LIN {X 0,Y 688.4,Z 749.56,A -85,B 0,C 180,E1 4160.047,E2 4160.047} C_VEL
LIN {X 0,Y 687.145,Z 749.56,A -85,B 0,C 180,E1 4160.767,E2 4160.767} C_VEL
LIN {X 0,Y 680.483,Z 749.56,A -85,B 0,C 180,E1 4162.72,E2 4162.72} C_VEL
LIN {X 0,Y 680.39,Z 749.56,A -85,B 0,C 180,E1 4162.905,E2 4162.905} C_VEL
LIN {X 0,Y 680.421,Z 749.56,A -85,B 0,C 180,E1 4167.797,E2 4167.797} C_VEL
LIN {X 0,Y 680.331,Z 749.56,A -85,B 0,C 180,E1 4172.429,E2 4172.429} C_VEL
LIN {X 0,Y 680.255,Z 749.56,A -85,B 0,C 180,E1 4176.897,E2 4176.897} C_VEL
LIN {X 0,Y 680.389,Z 749.56,A -85,B 0,C 180,E1 4182.867,E2 4182.867} C_VEL
LIN {X 0,Y 680.257,Z 749.803,A -85,B 0,C 180,E1 4188.162,E2 4188.162} C_VEL
LIN {X 0,Y 684.994,Z 759.606,A -85,B 0,C 180,E1 4188.65,E2 4188.65} C_VEL
LIN {X 0,Y 698.353,Z 783.089,A -85,B 0,C 180,E1 4189.918,E2 4189.918} C_VEL
LIN {X 0,Y 697.598,Z 850.093,A -85,B 0,C 180,E1 4190.892,E2 4190.892} C_VEL
LIN {X 0,Y 695.833,Z 894.125,A -85,B 0,C 180,E1 4191.958,E2 4191.958} C_VEL
LIN {X 0,Y 693.647,Z 941.776,A -85,B 0,C 180,E1 4193.674,E2 4193.674} C_VEL
LIN {X 0,Y 691.134,Z 988.011,A -85,B 0,C 180,E1 4195.911,E2 4195.911} C_VEL
LIN {X 0,Y 688.572,Z 1030.029,A -85,B 0,C 180,E1 4198.54,E2 4198.54} C_VEL
LIN {X 0,Y 686.252,Z 1069.067,A -85,B 0,C 180,E1 4201.577,E2 4201.577} C_VEL
LIN {X 0,Y 684.111,Z 1106.115,A -85,B 0,C 180,E1 4205.184,E2 4205.184} C_VEL
LIN {X 0,Y 682.717,Z 1135.913,A -85,B 0,C 180,E1 4208.795,E2 4208.795} C_VEL
LIN {X 0,Y 681.777,Z 1162.143,A -85,B 0,C 180,E1 4212.802,E2 4212.802} C_VEL
LIN {X 0,Y 681.145,Z 1182.346,A -85,B 0,C 180,E1 4216.855,E2 4216.855} C_VEL
LIN {X 0,Y 680.941,Z 1196.276,A -85,B 0,C 180,E1 4220.7,E2 4220.7} C_VEL
LIN {X 0,Y 680.837,Z 1204.797,A -85,B 0,C 180,E1 4224.267,E2 4224.267} C_VEL
LIN {X 0,Y 680.8,Z 1208.952,A -85,B 0,C 180,E1 4227.455,E2 4227.455} C_VEL
LIN {X 0,Y 680.945,Z 1209.669,A -85,B 0,C 180,E1 4231.271,E2 4231.271} C_VEL
LIN {X 0,Y 680.757,Z 1205.912,A -85,B 0,C 180,E1 4235.093,E2 4235.093} C_VEL
LIN {X 0,Y 680.821,Z 1197.333,A -85,B 0,C 180,E1 4238.938,E2 4238.938} C_VEL
LIN {X 0,Y 680.999,Z 1185.052,A -85,B 0,C 180,E1 4242.495,E2 4242.495} C_VEL
LIN {X 0,Y 681.502,Z 1166.472,A -85,B 0,C 180,E1 4246.421,E2 4246.421} C_VEL
LIN {X 0,Y 682.336,Z 1143.81,A -85,B 0,C 180,E1 4250.111,E2 4250.111} C_VEL
LIN {X 0,Y 683.774,Z 1113.746,A -85,B 0,C 180,E1 4253.958,E2 4253.958} C_VEL
LIN {X 0,Y 685.541,Z 1080.468,A -85,B 0,C 180,E1 4257.394,E2 4257.394} C_VEL
LIN {X 0,Y 687.949,Z 1040.284,A -85,B 0,C 180,E1 4260.73,E2 4260.73} C_VEL
LIN {X 0,Y 690.402,Z 998.657,A -85,B 0,C 180,E1 4263.478,E2 4263.478} C_VEL
LIN {X 0,Y 693.13,Z 953.433,A -85,B 0,C 180,E1 4265.821,E2 4265.821} C_VEL
LIN {X 0,Y 695.261,Z 909.712,A -85,B 0,C 180,E1 4267.534,E2 4267.534} C_VEL
LIN {X 0,Y 696.967,Z 867.67,A -85,B 0,C 180,E1 4268.733,E2 4268.733} C_VEL
LIN {X 0,Y 698.111,Z 822.718,A -85,B 0,C 180,E1 4269.568,E2 4269.568} C_VEL
LIN {X 0,Y 697.756,Z 782.473,A -85,B 0,C 180,E1 4270.132,E2 4270.132} C_VEL
LIN {X 0,Y 680.589,Z 751.281,A -85,B 0,C 180,E1 4271.792,E2 4271.792} C_VEL
LIN {X 0,Y 680.389,Z 749.56,A -85,B 0,C 180,E1 4271.887,E2 4271.887} C_VEL
LIN {X 0,Y 680.266,Z 749.56,A -85,B 0,C 180,E1 4276.482,E2 4276.482} C_VEL
LIN {X 0,Y 680.222,Z 749.56,A -85,B 0,C 180,E1 4281.539,E2 4281.539} C_VEL
LIN {X 0,Y 680.183,Z 749.56,A -85,B 0,C 180,E1 4286.264,E2 4286.264} C_VEL
LIN {X 0,Y 680.22,Z 749.56,A -85,B 0,C 180,E1 4290.746,E2 4290.746} C_VEL
LIN {X 0,Y 680.282,Z 749.56,A -85,B 0,C 180,E1 4295.607,E2 4295.607} C_VEL
LIN {X 0,Y 680.357,Z 749.56,A -85,B 0,C 180,E1 4300.542,E2 4300.542} C_VEL
LIN {X 0,Y 680.522,Z 749.56,A -85,B 0,C 180,E1 4305.865,E2 4305.865} C_VEL
LIN {X 0,Y 680.663,Z 749.56,A -85,B 0,C 180,E1 4311.063,E2 4311.063} C_VEL
LIN {X 0,Y 680.71,Z 749.56,A -85,B 0,C 180,E1 4316.185,E2 4316.185} C_VEL
LIN {X 0,Y 680.718,Z 749.56,A -85,B 0,C 180,E1 4320.004,E2 4320.004} C_VEL
LIN {X 0,Y 680.625,Z 749.56,A -85,B 0,C 180,E1 4325.099,E2 4325.099} C_VEL
LIN {X 0,Y 680.622,Z 749.56,A -85,B 0,C 180,E1 4330.235,E2 4330.235} C_VEL
LIN {X 0,Y 680.3,Z 749.56,A -85,B 0,C 180,E1 4335.463,E2 4335.463} C_VEL
LIN {X 0,Y 680.262,Z 749.56,A -85,B 0,C 180,E1 4341.097,E2 4341.097} C_VEL
LIN {X 0,Y 680.207,Z 749.56,A -85,B 0,C 180,E1 4346.384,E2 4346.384} C_VEL
LIN {X 0,Y 680.221,Z 749.56,A -85,B 0,C 180,E1 4350.732,E2 4350.732} C_VEL
LIN {X 0,Y 680.223,Z 749.56,A -85,B 0,C 180,E1 4355.287,E2 4355.287} C_VEL
LIN {X 0,Y 680.229,Z 749.56,A -85,B 0,C 180,E1 4360.114,E2 4360.114} C_VEL
LIN {X 0,Y 680.28,Z 749.714,A -85,B 0,C 180,E1 4363.859,E2 4363.859} C_VEL
LIN {X 0,Y 687.051,Z 763.886,A -85,B 0,C 180,E1 4364.465,E2 4364.465} C_VEL
LIN {X 0,Y 694.991,Z 780.667,A -85,B 0,C 180,E1 4365.184,E2 4365.184} C_VEL
LIN {X 0,Y 693.799,Z 827.247,A -85,B 0,C 180,E1 4366.107,E2 4366.107} C_VEL
LIN {X 0,Y 692.079,Z 873.368,A -85,B 0,C 180,E1 4367.568,E2 4367.568} C_VEL
LIN {X 0,Y 689.888,Z 916.339,A -85,B 0,C 180,E1 4369.457,E2 4369.457} C_VEL
LIN {X 0,Y 687.699,Z 958.747,A -85,B 0,C 180,E1 4371.915,E2 4371.915} C_VEL
LIN {X 0,Y 685.492,Z 998.587,A -85,B 0,C 180,E1 4374.891,E2 4374.891} C_VEL
LIN {X 0,Y 683.747,Z 1032.734,A -85,B 0,C 180,E1 4378.117,E2 4378.117} C_VEL
LIN {X 0,Y 682.43,Z 1061.896,A -85,B 0,C 180,E1 4381.571,E2 4381.571} C_VEL
LIN {X 0,Y 681.515,Z 1087.051,A -85,B 0,C 180,E1 4385.392,E2 4385.392} C_VEL
LIN {X 0,Y 681.141,Z 1103.808,A -85,B 0,C 180,E1 4388.727,E2 4388.727} C_VEL
LIN {X 0,Y 680.802,Z 1117.989,A -85,B 0,C 180,E1 4392.655,E2 4392.655} C_VEL
LIN {X 0,Y 680.792,Z 1125.467,A -85,B 0,C 180,E1 4395.868,E2 4395.868} C_VEL
LIN {X 0,Y 680.667,Z 1129.693,A -85,B 0,C 180,E1 4399.77,E2 4399.77} C_VEL
LIN {X 0,Y 680.816,Z 1128.697,A -85,B 0,C 180,E1 4403.629,E2 4403.629} C_VEL
LIN {X 0,Y 680.837,Z 1122.652,A -85,B 0,C 180,E1 4407.456,E2 4407.456} C_VEL
LIN {X 0,Y 680.918,Z 1111.397,A -85,B 0,C 180,E1 4411.272,E2 4411.272} C_VEL
LIN {X 0,Y 681.281,Z 1096.404,A -85,B 0,C 180,E1 4414.772,E2 4414.772} C_VEL
LIN {X 0,Y 681.915,Z 1075.181,A -85,B 0,C 180,E1 4418.443,E2 4418.443} C_VEL
LIN {X 0,Y 682.954,Z 1049.025,A -85,B 0,C 180,E1 4421.973,E2 4421.973} C_VEL
LIN {X 0,Y 684.646,Z 1014.871,A -85,B 0,C 180,E1 4425.577,E2 4425.577} C_VEL
LIN {X 0,Y 686.685,Z 976.797,A -85,B 0,C 180,E1 4428.732,E2 4428.732} C_VEL
LIN {X 0,Y 688.86,Z 937.867,A -85,B 0,C 180,E1 4431.278,E2 4431.278} C_VEL
LIN {X 0,Y 691.074,Z 895.773,A -85,B 0,C 180,E1 4433.426,E2 4433.426} C_VEL
LIN {X 0,Y 692.994,Z 852.505,A -85,B 0,C 180,E1 4435.065,E2 4435.065} C_VEL
LIN {X 0,Y 694.484,Z 807.428,A -85,B 0,C 180,E1 4436.259,E2 4436.259} C_VEL
LIN {X 0,Y 694.58,Z 779.374,A -85,B 0,C 180,E1 4436.77,E2 4436.77} C_VEL
LIN {X 0,Y 680.489,Z 750.957,A -85,B 0,C 180,E1 4438.022,E2 4438.022} C_VEL
LIN {X 0,Y 680.342,Z 749.56,A -85,B 0,C 180,E1 4438.085,E2 4438.085} C_VEL
LIN {X 0,Y 680.265,Z 749.56,A -85,B 0,C 180,E1 4443.735,E2 4443.735} C_VEL
LIN {X 0,Y 680.155,Z 749.56,A -85,B 0,C 180,E1 4448.951,E2 4448.951} C_VEL
LIN {X 0,Y 680.399,Z 749.56,A -85,B 0,C 180,E1 4453.512,E2 4453.512} C_VEL
LIN {X 0,Y 680.181,Z 749.56,A -85,B 0,C 180,E1 4459.058,E2 4459.058} C_VEL
LIN {X 0,Y 680.219,Z 749.56,A -85,B 0,C 180,E1 4463.138,E2 4463.138} C_VEL
LIN {X 0,Y 680.157,Z 749.56,A -85,B 0,C 180,E1 4467.772,E2 4467.772} C_VEL
LIN {X 0,Y 680.239,Z 749.56,A -85,B 0,C 180,E1 4472.698,E2 4472.698} C_VEL
LIN {X 0,Y 680.175,Z 749.56,A -85,B 0,C 180,E1 4477.805,E2 4477.805} C_VEL
LIN {X 0,Y 680.129,Z 749.56,A -85,B 0,C 180,E1 4482.823,E2 4482.823} C_VEL
LIN {X 0,Y 680.461,Z 749.56,A -85,B 0,C 180,E1 4487.724,E2 4487.724} C_VEL
LIN {X 0,Y 680.693,Z 749.56,A -85,B 0,C 180,E1 4492.342,E2 4492.342} C_VEL
LIN {X 0,Y 680.789,Z 749.56,A -85,B 0,C 180,E1 4497.452,E2 4497.452} C_VEL
LIN {X 0,Y 680.649,Z 749.56,A -85,B 0,C 180,E1 4502.541,E2 4502.541} C_VEL
LIN {X 0,Y 680.615,Z 749.56,A -85,B 0,C 180,E1 4506.37,E2 4506.37} C_VEL
LIN {X 0,Y 680.53,Z 749.56,A -85,B 0,C 180,E1 4511.525,E2 4511.525} C_VEL
LIN {X 0,Y 680.581,Z 749.56,A -85,B 0,C 180,E1 4516.774,E2 4516.774} C_VEL
LIN {X 0,Y 680.445,Z 749.56,A -85,B 0,C 180,E1 4522.178,E2 4522.178} C_VEL
LIN {X 0,Y 680.39,Z 749.56,A -85,B 0,C 180,E1 4522.905,E2 4522.905} C_VEL
LIN {X 0,Y 676.44,Z 749.56,A -85,B 0,C 180,E1 4524.339,E2 4524.339} C_VEL
LIN {X 0,Y 672.491,Z 749.56,A -85,B 0,C 180,E1 4525.789,E2 4525.789} C_VEL
LIN {X 0,Y 672.379,Z 749.56,A -85,B 0,C 180,E1 4531.347,E2 4531.347} C_VEL
LIN {X 0,Y 672.337,Z 749.56,A -85,B 0,C 180,E1 4535.988,E2 4535.988} C_VEL
LIN {X 0,Y 672.281,Z 749.56,A -85,B 0,C 180,E1 4540.678,E2 4540.678} C_VEL
LIN {X 0,Y 672.404,Z 749.56,A -85,B 0,C 180,E1 4545.981,E2 4545.981} C_VEL
LIN {X 0,Y 672.318,Z 749.803,A -85,B 0,C 180,E1 4547.554,E2 4547.554} C_VEL
LIN {X 0,Y 674.866,Z 755.349,A -85,B 0,C 180,E1 4547.829,E2 4547.829} C_VEL
LIN {X 0,Y 692.164,Z 785.898,A -85,B 0,C 180,E1 4549.523,E2 4549.523} C_VEL
LIN {X 0,Y 691.411,Z 851.6,A -85,B 0,C 180,E1 4550.506,E2 4550.506} C_VEL
LIN {X 0,Y 689.52,Z 895.054,A -85,B 0,C 180,E1 4551.576,E2 4551.576} C_VEL
LIN {X 0,Y 687.082,Z 942.72,A -85,B 0,C 180,E1 4553.314,E2 4553.314} C_VEL
LIN {X 0,Y 684.338,Z 988.281,A -85,B 0,C 180,E1 4555.54,E2 4555.54} C_VEL
LIN {X 0,Y 681.494,Z 1030.32,A -85,B 0,C 180,E1 4558.197,E2 4558.197} C_VEL
LIN {X 0,Y 678.955,Z 1069.071,A -85,B 0,C 180,E1 4561.243,E2 4561.243} C_VEL
LIN {X 0,Y 676.611,Z 1106.113,A -85,B 0,C 180,E1 4564.89,E2 4564.89} C_VEL
LIN {X 0,Y 675.023,Z 1136.317,A -85,B 0,C 180,E1 4568.598,E2 4568.598} C_VEL
LIN {X 0,Y 673.984,Z 1162.44,A -85,B 0,C 180,E1 4572.648,E2 4572.648} C_VEL
LIN {X 0,Y 673.306,Z 1182.347,A -85,B 0,C 180,E1 4576.7,E2 4576.7} C_VEL
LIN {X 0,Y 673.083,Z 1195.433,A -85,B 0,C 180,E1 4580.306,E2 4580.306} C_VEL
LIN {X 0,Y 672.955,Z 1204.795,A -85,B 0,C 180,E1 4584.2,E2 4584.2} C_VEL
LIN {X 0,Y 672.921,Z 1208.949,A -85,B 0,C 180,E1 4587.425,E2 4587.425} C_VEL
LIN {X 0,Y 673.045,Z 1209.669,A -85,B 0,C 180,E1 4591.286,E2 4591.286} C_VEL
LIN {X 0,Y 672.859,Z 1205.912,A -85,B 0,C 180,E1 4595.153,E2 4595.153} C_VEL
LIN {X 0,Y 672.96,Z 1197.333,A -85,B 0,C 180,E1 4599.043,E2 4599.043} C_VEL
LIN {X 0,Y 673.171,Z 1183.704,A -85,B 0,C 180,E1 4602.972,E2 4602.972} C_VEL
LIN {X 0,Y 673.827,Z 1164.715,A -85,B 0,C 180,E1 4606.949,E2 4606.949} C_VEL
LIN {X 0,Y 674.869,Z 1139.247,A -85,B 0,C 180,E1 4610.993,E2 4610.993} C_VEL
LIN {X 0,Y 676.475,Z 1109.315,A -85,B 0,C 180,E1 4614.761,E2 4614.761} C_VEL
LIN {X 0,Y 678.707,Z 1072.626,A -85,B 0,C 180,E1 4618.432,E2 4618.432} C_VEL
LIN {X 0,Y 681.195,Z 1035.134,A -85,B 0,C 180,E1 4621.46,E2 4621.46} C_VEL
LIN {X 0,Y 684.014,Z 991.951,A -85,B 0,C 180,E1 4624.252,E2 4624.252} C_VEL
LIN {X 0,Y 686.772,Z 948.289,A -85,B 0,C 180,E1 4626.447,E2 4626.447} C_VEL
LIN {X 0,Y 689.265,Z 900.278,A -85,B 0,C 180,E1 4628.256,E2 4628.256} C_VEL
LIN {X 0,Y 691.183,Z 852.976,A -85,B 0,C 180,E1 4629.48,E2 4629.48} C_VEL
LIN {X 0,Y 691.817,Z 785.747,A -85,B 0,C 180,E1 4630.504,E2 4630.504} C_VEL
LIN {X 0,Y 672.601,Z 751.041,A -85,B 0,C 180,E1 4632.407,E2 4632.407} C_VEL
LIN {X 0,Y 672.492,Z 749.56,A -85,B 0,C 180,E1 4632.493,E2 4632.493} C_VEL
LIN {X 0,Y 672.272,Z 749.56,A -85,B 0,C 180,E1 4637.882,E2 4637.882} C_VEL
LIN {X 0,Y 672.298,Z 749.56,A -85,B 0,C 180,E1 4642.639,E2 4642.639} C_VEL
LIN {X 0,Y 672.266,Z 749.56,A -85,B 0,C 180,E1 4647.355,E2 4647.355} C_VEL
LIN {X 0,Y 672.32,Z 749.56,A -85,B 0,C 180,E1 4651.839,E2 4651.839} C_VEL
LIN {X 0,Y 672.333,Z 749.56,A -85,B 0,C 180,E1 4657.146,E2 4657.146} C_VEL
LIN {X 0,Y 672.476,Z 749.56,A -85,B 0,C 180,E1 4661.667,E2 4661.667} C_VEL
LIN {X 0,Y 672.663,Z 749.56,A -85,B 0,C 180,E1 4667.021,E2 4667.021} C_VEL
LIN {X 0,Y 672.723,Z 749.56,A -85,B 0,C 180,E1 4672.258,E2 4672.258} C_VEL
LIN {X 0,Y 672.808,Z 749.56,A -85,B 0,C 180,E1 4676.14,E2 4676.14} C_VEL
LIN {X 0,Y 672.823,Z 749.56,A -85,B 0,C 180,E1 4680.004,E2 4680.004} C_VEL
LIN {X 0,Y 672.827,Z 749.56,A -85,B 0,C 180,E1 4683.867,E2 4683.867} C_VEL
LIN {X 0,Y 672.684,Z 749.56,A -85,B 0,C 180,E1 4689.051,E2 4689.051} C_VEL
LIN {X 0,Y 672.465,Z 749.56,A -85,B 0,C 180,E1 4694.315,E2 4694.315} C_VEL
LIN {X 0,Y 672.38,Z 749.56,A -85,B 0,C 180,E1 4699.705,E2 4699.705} C_VEL
LIN {X 0,Y 672.257,Z 749.56,A -85,B 0,C 180,E1 4705.288,E2 4705.288} C_VEL
LIN {X 0,Y 672.301,Z 749.56,A -85,B 0,C 180,E1 4709.641,E2 4709.641} C_VEL
LIN {X 0,Y 672.296,Z 749.56,A -85,B 0,C 180,E1 4714.194,E2 4714.194} C_VEL
LIN {X 0,Y 672.345,Z 749.56,A -85,B 0,C 180,E1 4719.005,E2 4719.005} C_VEL
LIN {X 0,Y 672.312,Z 749.56,A -85,B 0,C 180,E1 4723.34,E2 4723.34} C_VEL
LIN {X 0,Y 676.815,Z 759.567,A -85,B 0,C 180,E1 4723.765,E2 4723.765} C_VEL
LIN {X 0,Y 688.564,Z 782.52,A -85,B 0,C 180,E1 4724.825,E2 4724.825} C_VEL
LIN {X 0,Y 687.23,Z 828.392,A -85,B 0,C 180,E1 4725.759,E2 4725.759} C_VEL
LIN {X 0,Y 685.332,Z 874.495,A -85,B 0,C 180,E1 4727.239,E2 4727.239} C_VEL
LIN {X 0,Y 682.895,Z 917.839,A -85,B 0,C 180,E1 4729.179,E2 4729.179} C_VEL
LIN {X 0,Y 680.516,Z 959.618,A -85,B 0,C 180,E1 4731.642,E2 4731.642} C_VEL
LIN {X 0,Y 678.036,Z 1000.415,A -85,B 0,C 180,E1 4734.738,E2 4734.738} C_VEL
LIN {X 0,Y 676.02,Z 1035.648,A -85,B 0,C 180,E1 4738.158,E2 4738.158} C_VEL
LIN {X 0,Y 674.614,Z 1064.21,A -85,B 0,C 180,E1 4741.661,E2 4741.661} C_VEL
LIN {X 0,Y 673.684,Z 1088.271,A -85,B 0,C 180,E1 4745.42,E2 4745.42} C_VEL
LIN {X 0,Y 673.17,Z 1106.738,A -85,B 0,C 180,E1 4749.296,E2 4749.296} C_VEL
LIN {X 0,Y 672.881,Z 1119.377,A -85,B 0,C 180,E1 4753.026,E2 4753.026} C_VEL
LIN {X 0,Y 672.845,Z 1126.427,A -85,B 0,C 180,E1 4756.361,E2 4756.361} C_VEL
LIN {X 0,Y 672.771,Z 1129.664,A -85,B 0,C 180,E1 4759.649,E2 4759.649} C_VEL
LIN {X 0,Y 672.909,Z 1128.781,A -85,B 0,C 180,E1 4763.554,E2 4763.554} C_VEL
LIN {X 0,Y 672.968,Z 1122.908,A -85,B 0,C 180,E1 4767.427,E2 4767.427} C_VEL
LIN {X 0,Y 673.046,Z 1111.775,A -85,B 0,C 180,E1 4771.287,E2 4771.287} C_VEL
LIN {X 0,Y 673.417,Z 1096.913,A -85,B 0,C 180,E1 4774.828,E2 4774.828} C_VEL
LIN {X 0,Y 674.114,Z 1075.897,A -85,B 0,C 180,E1 4778.541,E2 4778.541} C_VEL
LIN {X 0,Y 675.248,Z 1049.936,A -85,B 0,C 180,E1 4782.111,E2 4782.111} C_VEL
LIN {X 0,Y 677.043,Z 1017.091,A -85,B 0,C 180,E1 4785.65,E2 4785.65} C_VEL
LIN {X 0,Y 679.171,Z 981.604,A -85,B 0,C 180,E1 4788.689,E2 4788.689} C_VEL
LIN {X 0,Y 681.648,Z 942.01,A -85,B 0,C 180,E1 4791.382,E2 4791.382} C_VEL
LIN {X 0,Y 684.033,Z 899.754,A -85,B 0,C 180,E1 4793.604,E2 4793.604} C_VEL
LIN {X 0,Y 686.094,Z 858.301,A -85,B 0,C 180,E1 4795.257,E2 4795.257} C_VEL
LIN {X 0,Y 687.88,Z 810.271,A -85,B 0,C 180,E1 4796.579,E2 4796.579} C_VEL
LIN {X 0,Y 688.21,Z 782.176,A -85,B 0,C 180,E1 4797.111,E2 4797.111} C_VEL
LIN {X 0,Y 672.466,Z 749.56,A -85,B 0,C 180,E1 4798.591,E2 4798.591} C_VEL
LIN {X 0,Y 672.361,Z 749.56,A -85,B 0,C 180,E1 4804.186,E2 4804.186} C_VEL
LIN {X 0,Y 672.263,Z 749.56,A -85,B 0,C 180,E1 4809.006,E2 4809.006} C_VEL
LIN {X 0,Y 672.472,Z 749.56,A -85,B 0,C 180,E1 4814.156,E2 4814.156} C_VEL
LIN {X 0,Y 672.343,Z 749.56,A -85,B 0,C 180,E1 4819.834,E2 4819.834} C_VEL
LIN {X 0,Y 672.271,Z 749.56,A -85,B 0,C 180,E1 4824.232,E2 4824.232} C_VEL
LIN {X 0,Y 672.243,Z 749.56,A -85,B 0,C 180,E1 4828.863,E2 4828.863} C_VEL
LIN {X 0,Y 672.275,Z 749.56,A -85,B 0,C 180,E1 4834.043,E2 4834.043} C_VEL
LIN {X 0,Y 672.343,Z 749.56,A -85,B 0,C 180,E1 4838.919,E2 4838.919} C_VEL
LIN {X 0,Y 672.385,Z 749.56,A -85,B 0,C 180,E1 4844.35,E2 4844.35} C_VEL
LIN {X 0,Y 672.729,Z 749.56,A -85,B 0,C 180,E1 4849.644,E2 4849.644} C_VEL
LIN {X 0,Y 672.728,Z 749.56,A -85,B 0,C 180,E1 4854.841,E2 4854.841} C_VEL
LIN {X 0,Y 672.851,Z 749.56,A -85,B 0,C 180,E1 4859.996,E2 4859.996} C_VEL
LIN {X 0,Y 672.882,Z 749.56,A -85,B 0,C 180,E1 4865.15,E2 4865.15} C_VEL
LIN {X 0,Y 672.67,Z 749.56,A -85,B 0,C 180,E1 4870.35,E2 4870.35} C_VEL
LIN {X 0,Y 672.661,Z 749.56,A -85,B 0,C 180,E1 4875.636,E2 4875.636} C_VEL
LIN {X 0,Y 672.594,Z 749.56,A -85,B 0,C 180,E1 4881.065,E2 4881.065} C_VEL
LIN {X 0,Y 672.491,Z 749.56,A -85,B 0,C 180,E1 4885.789,E2 4885.789} C_VEL
LIN {X 0,Y 671.256,Z 749.56,A -85,B 0,C 180,E1 4886.527,E2 4886.527} C_VEL
LIN {X 0,Y 664.616,Z 749.56,A -85,B 0,C 180,E1 4888.532,E2 4888.532} C_VEL
LIN {X 0,Y 664.498,Z 749.56,A -85,B 0,C 180,E1 4888.721,E2 4888.721} C_VEL
LIN {X 0,Y 664.529,Z 749.56,A -85,B 0,C 180,E1 4893.073,E2 4893.073} C_VEL
LIN {X 0,Y 664.37,Z 749.56,A -85,B 0,C 180,E1 4897.885,E2 4897.885} C_VEL
LIN {X 0,Y 664.493,Z 749.56,A -85,B 0,C 180,E1 4903.304,E2 4903.304} C_VEL
LIN {X 0,Y 664.428,Z 749.803,A -85,B 0,C 180,E1 4906.928,E2 4906.928} C_VEL
LIN {X 0,Y 667.032,Z 755.395,A -85,B 0,C 180,E1 4907.217,E2 4907.217} C_VEL
LIN {X 0,Y 686.149,Z 789.017,A -85,B 0,C 180,E1 4909.135,E2 4909.135} C_VEL
LIN {X 0,Y 685.237,Z 852.824,A -85,B 0,C 180,E1 4910.106,E2 4910.106} C_VEL
LIN {X 0,Y 683.131,Z 897.169,A -85,B 0,C 180,E1 4911.225,E2 4911.225} C_VEL
LIN {X 0,Y 680.403,Z 945.663,A -85,B 0,C 180,E1 4913.032,E2 4913.032} C_VEL
LIN {X 0,Y 677.474,Z 989.991,A -85,B 0,C 180,E1 4915.247,E2 4915.247} C_VEL
LIN {X 0,Y 674.297,Z 1033.297,A -85,B 0,C 180,E1 4918.042,E2 4918.042} C_VEL
LIN {X 0,Y 671.543,Z 1071.067,A -85,B 0,C 180,E1 4921.087,E2 4921.087} C_VEL
LIN {X 0,Y 668.981,Z 1108.342,A -85,B 0,C 180,E1 4924.834,E2 4924.834} C_VEL
LIN {X 0,Y 667.246,Z 1138.185,A -85,B 0,C 180,E1 4928.603,E2 4928.603} C_VEL
LIN {X 0,Y 666.176,Z 1163.173,A -85,B 0,C 180,E1 4932.567,E2 4932.567} C_VEL
LIN {X 0,Y 665.489,Z 1182.348,A -85,B 0,C 180,E1 4936.54,E2 4936.54} C_VEL
LIN {X 0,Y 665.216,Z 1195.43,A -85,B 0,C 180,E1 4940.19,E2 4940.19} C_VEL
LIN {X 0,Y 665.075,Z 1204.793,A -85,B 0,C 180,E1 4944.131,E2 4944.131} C_VEL
LIN {X 0,Y 665.017,Z 1208.946,A -85,B 0,C 180,E1 4947.395,E2 4947.395} C_VEL
LIN {X 0,Y 665.128,Z 1209.591,A -85,B 0,C 180,E1 4951.594,E2 4951.594} C_VEL
LIN {X 0,Y 665.034,Z 1204.796,A -85,B 0,C 180,E1 4955.868,E2 4955.868} C_VEL
LIN {X 0,Y 665.252,Z 1194.434,A -85,B 0,C 180,E1 4960.139,E2 4960.139} C_VEL
LIN {X 0,Y 665.566,Z 1179.548,A -85,B 0,C 180,E1 4964.126,E2 4964.126} C_VEL
LIN {X 0,Y 666.342,Z 1158.242,A -85,B 0,C 180,E1 4968.288,E2 4968.288} C_VEL
LIN {X 0,Y 667.632,Z 1132.551,A -85,B 0,C 180,E1 4972.181,E2 4972.181} C_VEL
LIN {X 0,Y 669.587,Z 1099.703,A -85,B 0,C 180,E1 4976.107,E2 4976.107} C_VEL
LIN {X 0,Y 672.02,Z 1064.38,A -85,B 0,C 180,E1 4979.497,E2 4979.497} C_VEL
LIN {X 0,Y 675.096,Z 1022.823,A -85,B 0,C 180,E1 4982.704,E2 4982.704} C_VEL
LIN {X 0,Y 678.185,Z 979.679,A -85,B 0,C 180,E1 4985.316,E2 4985.316} C_VEL
LIN {X 0,Y 681.196,Z 933.969,A -85,B 0,C 180,E1 4987.464,E2 4987.464} C_VEL
LIN {X 0,Y 683.687,Z 885.774,A -85,B 0,C 180,E1 4989.107,E2 4989.107} C_VEL
LIN {X 0,Y 685.602,Z 837.266,A -85,B 0,C 180,E1 4990.193,E2 4990.193} C_VEL
LIN {X 0,Y 685.817,Z 789.058,A -85,B 0,C 180,E1 4990.888,E2 4990.888} C_VEL
LIN {X 0,Y 664.767,Z 751.277,A -85,B 0,C 180,E1 4993.023,E2 4993.023} C_VEL
LIN {X 0,Y 664.572,Z 749.56,A -85,B 0,C 180,E1 4993.122,E2 4993.122} C_VEL
LIN {X 0,Y 664.33,Z 749.56,A -85,B 0,C 180,E1 4998.73,E2 4998.73} C_VEL
LIN {X 0,Y 664.391,Z 749.56,A -85,B 0,C 180,E1 5003.75,E2 5003.75} C_VEL
LIN {X 0,Y 664.363,Z 749.56,A -85,B 0,C 180,E1 5008.46,E2 5008.46} C_VEL
LIN {X 0,Y 664.419,Z 749.56,A -85,B 0,C 180,E1 5012.947,E2 5012.947} C_VEL
LIN {X 0,Y 664.451,Z 749.56,A -85,B 0,C 180,E1 5017.259,E2 5017.259} C_VEL
LIN {X 0,Y 664.648,Z 749.56,A -85,B 0,C 180,E1 5022.812,E2 5022.812} C_VEL
LIN {X 0,Y 664.719,Z 749.56,A -85,B 0,C 180,E1 5028.197,E2 5028.197} C_VEL
LIN {X 0,Y 664.802,Z 749.56,A -85,B 0,C 180,E1 5033.478,E2 5033.478} C_VEL
LIN {X 0,Y 665.082,Z 749.56,A -85,B 0,C 180,E1 5038.702,E2 5038.702} C_VEL
LIN {X 0,Y 664.937,Z 749.56,A -85,B 0,C 180,E1 5043.913,E2 5043.913} C_VEL
LIN {X 0,Y 664.774,Z 749.56,A -85,B 0,C 180,E1 5049.16,E2 5049.16} C_VEL
LIN {X 0,Y 664.555,Z 749.56,A -85,B 0,C 180,E1 5054.489,E2 5054.489} C_VEL
LIN {X 0,Y 664.452,Z 749.56,A -85,B 0,C 180,E1 5059.95,E2 5059.95} C_VEL
LIN {X 0,Y 664.349,Z 749.56,A -85,B 0,C 180,E1 5065.61,E2 5065.61} C_VEL
LIN {X 0,Y 664.349,Z 749.56,A -85,B 0,C 180,E1 5070.193,E2 5070.193} C_VEL
LIN {X 0,Y 664.325,Z 749.56,A -85,B 0,C 180,E1 5075.028,E2 5075.028} C_VEL
LIN {X 0,Y 664.419,Z 749.56,A -85,B 0,C 180,E1 5079.561,E2 5079.561} C_VEL
LIN {X 0,Y 664.411,Z 749.56,A -85,B 0,C 180,E1 5082.808,E2 5082.808} C_VEL
LIN {X 0,Y 668.851,Z 759.529,A -85,B 0,C 180,E1 5083.245,E2 5083.245} C_VEL
LIN {X 0,Y 682.166,Z 785.503,A -85,B 0,C 180,E1 5084.478,E2 5084.478} C_VEL
LIN {X 0,Y 680.573,Z 832.533,A -85,B 0,C 180,E1 5085.486,E2 5085.486} C_VEL
LIN {X 0,Y 678.538,Z 877.272,A -85,B 0,C 180,E1 5086.969,E2 5086.969} C_VEL
LIN {X 0,Y 675.768,Z 922.119,A -85,B 0,C 180,E1 5089.042,E2 5089.042} C_VEL
LIN {X 0,Y 673.154,Z 962.832,A -85,B 0,C 180,E1 5091.524,E2 5091.524} C_VEL
LIN {X 0,Y 670.664,Z 1000.702,A -85,B 0,C 180,E1 5094.453,E2 5094.453} C_VEL
LIN {X 0,Y 668.501,Z 1035.349,A -85,B 0,C 180,E1 5097.854,E2 5097.854} C_VEL
LIN {X 0,Y 666.954,Z 1063.482,A -85,B 0,C 180,E1 5101.327,E2 5101.327} C_VEL
LIN {X 0,Y 665.866,Z 1088.15,A -85,B 0,C 180,E1 5105.21,E2 5105.21} C_VEL
LIN {X 0,Y 665.316,Z 1106.268,A -85,B 0,C 180,E1 5109.04,E2 5109.04} C_VEL
LIN {X 0,Y 664.993,Z 1119.047,A -85,B 0,C 180,E1 5112.818,E2 5112.818} C_VEL
LIN {X 0,Y 664.963,Z 1126.279,A -85,B 0,C 180,E1 5116.196,E2 5116.196} C_VEL
LIN {X 0,Y 664.854,Z 1129.635,A -85,B 0,C 180,E1 5119.524,E2 5119.524} C_VEL
LIN {X 0,Y 665.001,Z 1128.866,A -85,B 0,C 180,E1 5123.477,E2 5123.477} C_VEL
LIN {X 0,Y 665.07,Z 1123.165,A -85,B 0,C 180,E1 5127.396,E2 5127.396} C_VEL
LIN {X 0,Y 665.176,Z 1112.153,A -85,B 0,C 180,E1 5131.302,E2 5131.302} C_VEL
LIN {X 0,Y 665.564,Z 1097.421,A -85,B 0,C 180,E1 5134.885,E2 5134.885} C_VEL
LIN {X 0,Y 666.314,Z 1076.606,A -85,B 0,C 180,E1 5138.642,E2 5138.642} C_VEL
LIN {X 0,Y 667.586,Z 1049.529,A -85,B 0,C 180,E1 5142.418,E2 5142.418} C_VEL
LIN {X 0,Y 669.718,Z 1015.818,A -85,B 0,C 180,E1 5146.068,E2 5146.068} C_VEL
LIN {X 0,Y 672.045,Z 979.415,A -85,B 0,C 180,E1 5149.183,E2 5149.183} C_VEL
LIN {X 0,Y 674.675,Z 940.793,A -85,B 0,C 180,E1 5151.805,E2 5151.805} C_VEL
LIN {X 0,Y 677.276,Z 899.302,A -85,B 0,C 180,E1 5153.994,E2 5153.994} C_VEL
LIN {X 0,Y 679.507,Z 858.279,A -85,B 0,C 180,E1 5155.637,E2 5155.637} C_VEL
LIN {X 0,Y 681.406,Z 810.884,A -85,B 0,C 180,E1 5156.955,E2 5156.955} C_VEL
LIN {X 0,Y 681.832,Z 785.206,A -85,B 0,C 180,E1 5157.458,E2 5157.458} C_VEL
LIN {X 0,Y 664.499,Z 749.56,A -85,B 0,C 180,E1 5159.121,E2 5159.121} C_VEL
LIN {X 0,Y 664.394,Z 749.56,A -85,B 0,C 180,E1 5164.654,E2 5164.654} C_VEL
LIN {X 0,Y 664.364,Z 749.56,A -85,B 0,C 180,E1 5169.56,E2 5169.56} C_VEL
LIN {X 0,Y 664.46,Z 749.56,A -85,B 0,C 180,E1 5174.831,E2 5174.831} C_VEL
LIN {X 0,Y 664.429,Z 749.56,A -85,B 0,C 180,E1 5180.649,E2 5180.649} C_VEL
LIN {X 0,Y 664.339,Z 749.56,A -85,B 0,C 180,E1 5185.338,E2 5185.338} C_VEL
LIN {X 0,Y 664.324,Z 749.56,A -85,B 0,C 180,E1 5189.967,E2 5189.967} C_VEL
LIN {X 0,Y 664.366,Z 749.56,A -85,B 0,C 180,E1 5194.39,E2 5194.39} C_VEL
LIN {X 0,Y 664.406,Z 749.56,A -85,B 0,C 180,E1 5200.048,E2 5200.048} C_VEL
LIN {X 0,Y 664.541,Z 749.56,A -85,B 0,C 180,E1 5205.511,E2 5205.511} C_VEL
LIN {X 0,Y 664.785,Z 749.56,A -85,B 0,C 180,E1 5210.84,E2 5210.84} C_VEL
LIN {X 0,Y 664.927,Z 749.56,A -85,B 0,C 180,E1 5216.087,E2 5216.087} C_VEL
LIN {X 0,Y 665.092,Z 749.56,A -85,B 0,C 180,E1 5221.364,E2 5221.364} C_VEL
LIN {X 0,Y 664.808,Z 749.56,A -85,B 0,C 180,E1 5226.522,E2 5226.522} C_VEL
LIN {X 0,Y 664.711,Z 749.56,A -85,B 0,C 180,E1 5231.803,E2 5231.803} C_VEL
LIN {X 0,Y 664.734,Z 749.56,A -85,B 0,C 180,E1 5237.294,E2 5237.294} C_VEL
LIN {X 0,Y 664.602,Z 749.56,A -85,B 0,C 180,E1 5242.736,E2 5242.736} C_VEL
LIN {X 0,Y 664.562,Z 749.56,A -85,B 0,C 180,E1 5247.524,E2 5247.524} C_VEL
LIN {X 0,Y 664.498,Z 749.56,A -85,B 0,C 180,E1 5248.721,E2 5248.721} C_VEL
LIN {X 0,Y 660.493,Z 749.56,A -85,B 0,C 180,E1 5250.196,E2 5250.196} C_VEL
LIN {X 0,Y 656.566,Z 749.56,A -85,B 0,C 180,E1 5251.688,E2 5251.688} C_VEL
LIN {X 0,Y 656.486,Z 749.56,A -85,B 0,C 180,E1 5256.758,E2 5256.758} C_VEL
LIN {X 0,Y 656.519,Z 749.56,A -85,B 0,C 180,E1 5262.56,E2 5262.56} C_VEL
LIN {X 0,Y 656.508,Z 749.817,A -85,B 0,C 180,E1 5266.279,E2 5266.279} C_VEL
LIN {X 0,Y 659.111,Z 755.392,A -85,B 0,C 180,E1 5266.577,E2 5266.577} C_VEL
LIN {X 0,Y 680.225,Z 792.246,A -85,B 0,C 180,E1 5268.746,E2 5268.746} C_VEL
LIN {X 0,Y 679.182,Z 852.919,A -85,B 0,C 180,E1 5269.68,E2 5269.68} C_VEL
LIN {X 0,Y 676.969,Z 896.038,A -85,B 0,C 180,E1 5270.763,E2 5270.763} C_VEL
LIN {X 0,Y 674.168,Z 942.933,A -85,B 0,C 180,E1 5272.502,E2 5272.502} C_VEL
LIN {X 0,Y 670.918,Z 988.257,A -85,B 0,C 180,E1 5274.748,E2 5274.748} C_VEL
LIN {X 0,Y 667.557,Z 1030.497,A -85,B 0,C 180,E1 5277.466,E2 5277.466} C_VEL
LIN {X 0,Y 664.382,Z 1070.127,A -85,B 0,C 180,E1 5280.653,E2 5280.653} C_VEL
LIN {X 0,Y 661.58,Z 1107.327,A -85,B 0,C 180,E1 5284.417,E2 5284.417} C_VEL
LIN {X 0,Y 659.662,Z 1137.131,A -85,B 0,C 180,E1 5288.192,E2 5288.192} C_VEL
LIN {X 0,Y 658.395,Z 1163.171,A -85,B 0,C 180,E1 5292.354,E2 5292.354} C_VEL
LIN {X 0,Y 657.679,Z 1182.349,A -85,B 0,C 180,E1 5296.378,E2 5296.378} C_VEL
LIN {X 0,Y 657.359,Z 1195.427,A -85,B 0,C 180,E1 5300.071,E2 5300.071} C_VEL
LIN {X 0,Y 657.186,Z 1204.79,A -85,B 0,C 180,E1 5304.06,E2 5304.06} C_VEL
LIN {X 0,Y 657.114,Z 1208.943,A -85,B 0,C 180,E1 5307.363,E2 5307.363} C_VEL
LIN {X 0,Y 657.268,Z 1209.668,A -85,B 0,C 180,E1 5311.317,E2 5311.317} C_VEL
LIN {X 0,Y 657.092,Z 1205.912,A -85,B 0,C 180,E1 5315.277,E2 5315.277} C_VEL
LIN {X 0,Y 657.191,Z 1197.333,A -85,B 0,C 180,E1 5319.262,E2 5319.262} C_VEL
LIN {X 0,Y 657.499,Z 1183.706,A -85,B 0,C 180,E1 5323.286,E2 5323.286} C_VEL
LIN {X 0,Y 658.323,Z 1164.718,A -85,B 0,C 180,E1 5327.361,E2 5327.361} C_VEL
LIN {X 0,Y 659.525,Z 1139.251,A -85,B 0,C 180,E1 5331.505,E2 5331.505} C_VEL
LIN {X 0,Y 661.477,Z 1109.999,A -85,B 0,C 180,E1 5335.28,E2 5335.28} C_VEL
LIN {X 0,Y 664.044,Z 1074.33,A -85,B 0,C 180,E1 5338.954,E2 5338.954} C_VEL
LIN {X 0,Y 666.975,Z 1037.132,A -85,B 0,C 180,E1 5342.057,E2 5342.057} C_VEL
LIN {X 0,Y 670.466,Z 992.954,A -85,B 0,C 180,E1 5344.979,E2 5344.979} C_VEL
LIN {X 0,Y 673.75,Z 948.295,A -85,B 0,C 180,E1 5347.269,E2 5347.269} C_VEL
LIN {X 0,Y 676.773,Z 898.533,A -85,B 0,C 180,E1 5349.159,E2 5349.159} C_VEL
LIN {X 0,Y 679.049,Z 850.539,A -85,B 0,C 180,E1 5350.381,E2 5350.381} C_VEL
LIN {X 0,Y 679.865,Z 792.31,A -85,B 0,C 180,E1 5351.279,E2 5351.279} C_VEL
LIN {X 0,Y 656.734,Z 750.944,A -85,B 0,C 180,E1 5353.686,E2 5353.686} C_VEL
LIN {X 0,Y 656.597,Z 749.56,A -85,B 0,C 180,E1 5353.777,E2 5353.777} C_VEL
LIN {X 0,Y 656.399,Z 749.56,A -85,B 0,C 180,E1 5359.437,E2 5359.437} C_VEL
LIN {X 0,Y 656.445,Z 749.56,A -85,B 0,C 180,E1 5364.869,E2 5364.869} C_VEL
LIN {X 0,Y 656.432,Z 749.56,A -85,B 0,C 180,E1 5369.576,E2 5369.576} C_VEL
LIN {X 0,Y 656.527,Z 749.56,A -85,B 0,C 180,E1 5374.07,E2 5374.07} C_VEL
LIN {X 0,Y 656.531,Z 749.56,A -85,B 0,C 180,E1 5378.394,E2 5378.394} C_VEL
LIN {X 0,Y 656.786,Z 749.56,A -85,B 0,C 180,E1 5383.976,E2 5383.976} C_VEL
LIN {X 0,Y 656.83,Z 749.56,A -85,B 0,C 180,E1 5389.398,E2 5389.398} C_VEL
LIN {X 0,Y 657.073,Z 749.56,A -85,B 0,C 180,E1 5394.725,E2 5394.725} C_VEL
LIN {X 0,Y 657.066,Z 749.56,A -85,B 0,C 180,E1 5400.004,E2 5400.004} C_VEL
LIN {X 0,Y 656.916,Z 749.56,A -85,B 0,C 180,E1 5405.283,E2 5405.283} C_VEL
LIN {X 0,Y 656.87,Z 749.56,A -85,B 0,C 180,E1 5410.609,E2 5410.609} C_VEL
LIN {X 0,Y 656.507,Z 749.56,A -85,B 0,C 180,E1 5416.038,E2 5416.038} C_VEL
LIN {X 0,Y 656.498,Z 749.56,A -85,B 0,C 180,E1 5421.615,E2 5421.615} C_VEL
LIN {X 0,Y 656.446,Z 749.56,A -85,B 0,C 180,E1 5427.418,E2 5427.418} C_VEL
LIN {X 0,Y 656.449,Z 749.56,A -85,B 0,C 180,E1 5431.974,E2 5431.974} C_VEL
LIN {X 0,Y 656.456,Z 749.56,A -85,B 0,C 180,E1 5436.769,E2 5436.769} C_VEL
LIN {X 0,Y 656.47,Z 749.56,A -85,B 0,C 180,E1 5442.237,E2 5442.237} C_VEL
LIN {X 0,Y 662.919,Z 763.316,A -85,B 0,C 180,E1 5442.899,E2 5442.899} C_VEL
LIN {X 0,Y 675.772,Z 788.611,A -85,B 0,C 180,E1 5444.129,E2 5444.129} C_VEL
LIN {X 0,Y 673.972,Z 835.446,A -85,B 0,C 180,E1 5445.173,E2 5445.173} C_VEL
LIN {X 0,Y 671.816,Z 878.224,A -85,B 0,C 180,E1 5446.625,E2 5446.625} C_VEL
LIN {X 0,Y 668.816,Z 923.568,A -85,B 0,C 180,E1 5448.753,E2 5448.753} C_VEL
LIN {X 0,Y 665.966,Z 963.997,A -85,B 0,C 180,E1 5451.261,E2 5451.261} C_VEL
LIN {X 0,Y 663.274,Z 1001.185,A -85,B 0,C 180,E1 5454.179,E2 5454.179} C_VEL
LIN {X 0,Y 660.828,Z 1037.386,A -85,B 0,C 180,E1 5457.797,E2 5457.797} C_VEL
LIN {X 0,Y 659.087,Z 1066.701,A -85,B 0,C 180,E1 5461.547,E2 5461.547} C_VEL
LIN {X 0,Y 658.033,Z 1089.296,A -85,B 0,C 180,E1 5465.24,E2 5465.24} C_VEL
LIN {X 0,Y 657.446,Z 1107.204,A -85,B 0,C 180,E1 5469.13,E2 5469.13} C_VEL
LIN {X 0,Y 657.138,Z 1118.719,A -85,B 0,C 180,E1 5472.607,E2 5472.607} C_VEL
LIN {X 0,Y 657.064,Z 1126.091,A -85,B 0,C 180,E1 5476.027,E2 5476.027} C_VEL
LIN {X 0,Y 656.937,Z 1129.606,A -85,B 0,C 180,E1 5479.397,E2 5479.397} C_VEL
LIN {X 0,Y 657.092,Z 1128.95,A -85,B 0,C 180,E1 5483.398,E2 5483.398} C_VEL
LIN {X 0,Y 657.171,Z 1123.391,A -85,B 0,C 180,E1 5487.365,E2 5487.365} C_VEL
LIN {X 0,Y 657.305,Z 1112.53,A -85,B 0,C 180,E1 5491.318,E2 5491.318} C_VEL
LIN {X 0,Y 657.763,Z 1096.422,A -85,B 0,C 180,E1 5495.273,E2 5495.273} C_VEL
LIN {X 0,Y 658.57,Z 1075.224,A -85,B 0,C 180,E1 5499.077,E2 5499.077} C_VEL
LIN {X 0,Y 659.988,Z 1049.093,A -85,B 0,C 180,E1 5502.732,E2 5502.732} C_VEL
LIN {X 0,Y 662.298,Z 1015.209,A -85,B 0,C 180,E1 5506.432,E2 5506.432} C_VEL
LIN {X 0,Y 664.862,Z 979.209,A -85,B 0,C 180,E1 5509.532,E2 5509.532} C_VEL
LIN {X 0,Y 667.742,Z 940.117,A -85,B 0,C 180,E1 5512.204,E2 5512.204} C_VEL
LIN {X 0,Y 670.539,Z 899.189,A -85,B 0,C 180,E1 5514.375,E2 5514.375} C_VEL
LIN {X 0,Y 672.983,Z 857.513,A -85,B 0,C 180,E1 5516.05,E2 5516.05} C_VEL
LIN {X 0,Y 675.052,Z 810.16,A -85,B 0,C 180,E1 5517.366,E2 5517.366} C_VEL
LIN {X 0,Y 675.285,Z 787.564,A -85,B 0,C 180,E1 5517.832,E2 5517.832} C_VEL
LIN {X 0,Y 656.565,Z 750.001,A -85,B 0,C 180,E1 5519.64,E2 5519.64} C_VEL
LIN {X 0,Y 656.493,Z 749.56,A -85,B 0,C 180,E1 5525.132,E2 5525.132} C_VEL
LIN {X 0,Y 656.42,Z 749.56,A -85,B 0,C 180,E1 5530.556,E2 5530.556} C_VEL
LIN {X 0,Y 656.475,Z 749.56,A -85,B 0,C 180,E1 5535.528,E2 5535.528} C_VEL
LIN {X 0,Y 656.428,Z 749.56,A -85,B 0,C 180,E1 5539.86,E2 5539.86} C_VEL
LIN {X 0,Y 656.423,Z 749.56,A -85,B 0,C 180,E1 5544.859,E2 5544.859} C_VEL
LIN {X 0,Y 656.403,Z 749.56,A -85,B 0,C 180,E1 5549.566,E2 5549.566} C_VEL
LIN {X 0,Y 656.429,Z 749.56,A -85,B 0,C 180,E1 5554.058,E2 5554.058} C_VEL
LIN {X 0,Y 656.497,Z 749.56,A -85,B 0,C 180,E1 5559.797,E2 5559.797} C_VEL
LIN {X 0,Y 656.607,Z 749.56,A -85,B 0,C 180,E1 5565.332,E2 5565.332} C_VEL
LIN {X 0,Y 656.887,Z 749.56,A -85,B 0,C 180,E1 5570.729,E2 5570.729} C_VEL
LIN {X 0,Y 657.017,Z 749.56,A -85,B 0,C 180,E1 5576.04,E2 5576.04} C_VEL
LIN {X 0,Y 657.225,Z 749.56,A -85,B 0,C 180,E1 5581.314,E2 5581.314} C_VEL
LIN {X 0,Y 656.9,Z 749.56,A -85,B 0,C 180,E1 5586.601,E2 5586.601} C_VEL
LIN {X 0,Y 656.805,Z 749.56,A -85,B 0,C 180,E1 5591.947,E2 5591.947} C_VEL
LIN {X 0,Y 656.838,Z 749.56,A -85,B 0,C 180,E1 5597.399,E2 5597.399} C_VEL
LIN {X 0,Y 656.68,Z 749.56,A -85,B 0,C 180,E1 5603.026,E2 5603.026} C_VEL
LIN {X 0,Y 656.658,Z 749.56,A -85,B 0,C 180,E1 5607.4,E2 5607.4} C_VEL
LIN {X 0,Y 656.566,Z 749.56,A -85,B 0,C 180,E1 5611.688,E2 5611.688} C_VEL
LIN {X 0,Y 652.569,Z 749.56,A -85,B 0,C 180,E1 5613.178,E2 5613.178} C_VEL
LIN {X 0,Y 648.577,Z 749.56,A -85,B 0,C 180,E1 5614.687,E2 5614.687} C_VEL
LIN {X 0,Y 648.473,Z 749.56,A -85,B 0,C 180,E1 5619.735,E2 5619.735} C_VEL
LIN {X 0,Y 648.649,Z 749.56,A -85,B 0,C 180,E1 5624.335,E2 5624.335} C_VEL
LIN {X 0,Y 648.633,Z 749.817,A -85,B 0,C 180,E1 5625.61,E2 5625.61} C_VEL
LIN {X 0,Y 651.228,Z 755.452,A -85,B 0,C 180,E1 5625.918,E2 5625.918} C_VEL
LIN {X 0,Y 674.298,Z 795.538,A -85,B 0,C 180,E1 5628.349,E2 5628.349} C_VEL
LIN {X 0,Y 673.124,Z 853.073,A -85,B 0,C 180,E1 5629.245,E2 5629.245} C_VEL
LIN {X 0,Y 670.707,Z 897.317,A -85,B 0,C 180,E1 5630.373,E2 5630.373} C_VEL
LIN {X 0,Y 667.69,Z 943.967,A -85,B 0,C 180,E1 5632.124,E2 5632.124} C_VEL
LIN {X 0,Y 664.24,Z 988.496,A -85,B 0,C 180,E1 5634.355,E2 5634.355} C_VEL
LIN {X 0,Y 660.649,Z 1030.376,A -85,B 0,C 180,E1 5637.074,E2 5637.074} C_VEL
LIN {X 0,Y 657.301,Z 1068.918,A -85,B 0,C 180,E1 5640.188,E2 5640.188} C_VEL
LIN {X 0,Y 654.208,Z 1106.106,A -85,B 0,C 180,E1 5643.967,E2 5643.967} C_VEL
LIN {X 0,Y 652.102,Z 1136.046,A -85,B 0,C 180,E1 5647.766,E2 5647.766} C_VEL
LIN {X 0,Y 650.647,Z 1162.441,A -85,B 0,C 180,E1 5652.006,E2 5652.006} C_VEL
LIN {X 0,Y 649.836,Z 1182.35,A -85,B 0,C 180,E1 5656.21,E2 5656.21} C_VEL
LIN {X 0,Y 649.477,Z 1195.424,A -85,B 0,C 180,E1 5659.95,E2 5659.95} C_VEL
LIN {X 0,Y 649.298,Z 1204.787,A -85,B 0,C 180,E1 5663.988,E2 5663.988} C_VEL
LIN {X 0,Y 649.231,Z 1208.94,A -85,B 0,C 180,E1 5667.331,E2 5667.331} C_VEL
LIN {X 0,Y 649.365,Z 1209.668,A -85,B 0,C 180,E1 5671.333,E2 5671.333} C_VEL
LIN {X 0,Y 649.215,Z 1205.912,A -85,B 0,C 180,E1 5675.342,E2 5675.342} C_VEL
LIN {X 0,Y 649.313,Z 1197.332,A -85,B 0,C 180,E1 5679.375,E2 5679.375} C_VEL
LIN {X 0,Y 649.689,Z 1183.707,A -85,B 0,C 180,E1 5683.449,E2 5683.449} C_VEL
LIN {X 0,Y 650.649,Z 1163.571,A -85,B 0,C 180,E1 5687.79,E2 5687.79} C_VEL
LIN {X 0,Y 652.042,Z 1137.428,A -85,B 0,C 180,E1 5692.033,E2 5692.033} C_VEL
LIN {X 0,Y 654.168,Z 1107.521,A -85,B 0,C 180,E1 5695.872,E2 5695.872} C_VEL
LIN {X 0,Y 657.111,Z 1070.869,A -85,B 0,C 180,E1 5699.63,E2 5699.63} C_VEL
LIN {X 0,Y 660.477,Z 1031.65,A -85,B 0,C 180,E1 5702.838,E2 5702.838} C_VEL
LIN {X 0,Y 664.212,Z 988.542,A -85,B 0,C 180,E1 5705.644,E2 5705.644} C_VEL
LIN {X 0,Y 667.689,Z 942.443,A -85,B 0,C 180,E1 5707.949,E2 5707.949} C_VEL
LIN {X 0,Y 670.893,Z 893.885,A -85,B 0,C 180,E1 5709.736,E2 5709.736} C_VEL
LIN {X 0,Y 673.194,Z 845.008,A -85,B 0,C 180,E1 5710.925,E2 5710.925} C_VEL
LIN {X 0,Y 673.737,Z 795.103,A -85,B 0,C 180,E1 5711.699,E2 5711.699} C_VEL
LIN {X 0,Y 650.299,Z 754.379,A -85,B 0,C 180,E1 5714.178,E2 5714.178} C_VEL
LIN {X 0,Y 648.67,Z 749.56,A -85,B 0,C 180,E1 5714.451,E2 5714.451} C_VEL
LIN {X 0,Y 648.481,Z 749.56,A -85,B 0,C 180,E1 5720.262,E2 5720.262} C_VEL
LIN {X 0,Y 648.534,Z 749.56,A -85,B 0,C 180,E1 5724.638,E2 5724.638} C_VEL
LIN {X 0,Y 648.55,Z 749.56,A -85,B 0,C 180,E1 5729.552,E2 5729.552} C_VEL
LIN {X 0,Y 648.622,Z 749.56,A -85,B 0,C 180,E1 5735.311,E2 5735.311} C_VEL
LIN {X 0,Y 648.713,Z 749.56,A -85,B 0,C 180,E1 5740.97,E2 5740.97} C_VEL
LIN {X 0,Y 648.874,Z 749.56,A -85,B 0,C 180,E1 5745.16,E2 5745.16} C_VEL
LIN {X 0,Y 649.006,Z 749.56,A -85,B 0,C 180,E1 5750.623,E2 5750.623} C_VEL
LIN {X 0,Y 649.14,Z 749.56,A -85,B 0,C 180,E1 5755.999,E2 5755.999} C_VEL
LIN {X 0,Y 649.179,Z 749.56,A -85,B 0,C 180,E1 5760.004,E2 5760.004} C_VEL
LIN {X 0,Y 649.137,Z 749.56,A -85,B 0,C 180,E1 5764.008,E2 5764.008} C_VEL
LIN {X 0,Y 648.962,Z 749.56,A -85,B 0,C 180,E1 5769.385,E2 5769.385} C_VEL
LIN {X 0,Y 648.724,Z 749.56,A -85,B 0,C 180,E1 5774.851,E2 5774.851} C_VEL
LIN {X 0,Y 648.62,Z 749.56,A -85,B 0,C 180,E1 5780.459,E2 5780.459} C_VEL
LIN {X 0,Y 648.492,Z 749.56,A -85,B 0,C 180,E1 5786.284,E2 5786.284} C_VEL
LIN {X 0,Y 648.538,Z 749.56,A -85,B 0,C 180,E1 5790.843,E2 5790.843} C_VEL
LIN {X 0,Y 648.523,Z 749.56,A -85,B 0,C 180,E1 5795.634,E2 5795.634} C_VEL
LIN {X 0,Y 648.531,Z 749.56,A -85,B 0,C 180,E1 5801.454,E2 5801.454} C_VEL
LIN {X 0,Y 648.555,Z 749.909,A -85,B 0,C 180,E1 5801.634,E2 5801.634} C_VEL
LIN {X 0,Y 655.968,Z 764.672,A -85,B 0,C 180,E1 5802.432,E2 5802.432} C_VEL
LIN {X 0,Y 669.398,Z 791.797,A -85,B 0,C 180,E1 5803.786,E2 5803.786} C_VEL
LIN {X 0,Y 667.451,Z 837.486,A -85,B 0,C 180,E1 5804.831,E2 5804.831} C_VEL
LIN {X 0,Y 665.02,Z 880.846,A -85,B 0,C 180,E1 5806.345,E2 5806.345} C_VEL
LIN {X 0,Y 661.755,Z 926.423,A -85,B 0,C 180,E1 5808.532,E2 5808.532} C_VEL
LIN {X 0,Y 658.412,Z 969.493,A -85,B 0,C 180,E1 5811.299,E2 5811.299} C_VEL
LIN {X 0,Y 655.631,Z 1005.55,A -85,B 0,C 180,E1 5814.262,E2 5814.262} C_VEL
LIN {X 0,Y 653.237,Z 1038.298,A -85,B 0,C 180,E1 5817.617,E2 5817.617} C_VEL
LIN {X 0,Y 651.365,Z 1067.379,A -85,B 0,C 180,E1 5821.408,E2 5821.408} C_VEL
LIN {X 0,Y 650.178,Z 1090.436,A -85,B 0,C 180,E1 5825.27,E2 5825.27} C_VEL
LIN {X 0,Y 649.564,Z 1108.482,A -85,B 0,C 180,E1 5829.31,E2 5829.31} C_VEL
LIN {X 0,Y 649.195,Z 1120.488,A -85,B 0,C 180,E1 5833.204,E2 5833.204} C_VEL
LIN {X 0,Y 649.15,Z 1126.871,A -85,B 0,C 180,E1 5836.54,E2 5836.54} C_VEL
LIN {X 0,Y 649.117,Z 1129.923,A -85,B 0,C 180,E1 5840.622,E2 5840.622} C_VEL
LIN {X 0,Y 649.195,Z 1127.782,A -85,B 0,C 180,E1 5844.658,E2 5844.658} C_VEL
LIN {X 0,Y 649.242,Z 1120.578,A -85,B 0,C 180,E1 5848.667,E2 5848.667} C_VEL
LIN {X 0,Y 649.517,Z 1109.508,A -85,B 0,C 180,E1 5852.334,E2 5852.334} C_VEL
LIN {X 0,Y 649.999,Z 1093.661,A -85,B 0,C 180,E1 5856.006,E2 5856.006} C_VEL
LIN {X 0,Y 651.17,Z 1070.645,A -85,B 0,C 180,E1 5860.024,E2 5860.024} C_VEL
LIN {X 0,Y 652.895,Z 1041.803,A -85,B 0,C 180,E1 5863.877,E2 5863.877} C_VEL
LIN {X 0,Y 655.232,Z 1011.012,A -85,B 0,C 180,E1 5867.14,E2 5867.14} C_VEL
LIN {X 0,Y 658.112,Z 973.466,A -85,B 0,C 180,E1 5870.323,E2 5870.323} C_VEL
LIN {X 0,Y 661.464,Z 930.816,A -85,B 0,C 180,E1 5873.12,E2 5873.12} C_VEL
LIN {X 0,Y 664.421,Z 889.565,A -85,B 0,C 180,E1 5875.197,E2 5875.197} C_VEL
LIN {X 0,Y 667.146,Z 845.195,A -85,B 0,C 180,E1 5876.844,E2 5876.844} C_VEL
LIN {X 0,Y 669.011,Z 803.693,A -85,B 0,C 180,E1 5877.904,E2 5877.904} C_VEL
LIN {X 0,Y 668.763,Z 790.243,A -85,B 0,C 180,E1 5878.198,E2 5878.198} C_VEL
LIN {X 0,Y 648.661,Z 750.369,A -85,B 0,C 180,E1 5880.249,E2 5880.249} C_VEL
LIN {X 0,Y 648.575,Z 749.56,A -85,B 0,C 180,E1 5884,E2 5884} C_VEL
LIN {X 0,Y 648.475,Z 749.56,A -85,B 0,C 180,E1 5889.729,E2 5889.729} C_VEL
LIN {X 0,Y 648.639,Z 749.56,A -85,B 0,C 180,E1 5894.34,E2 5894.34} C_VEL
LIN {X 0,Y 648.497,Z 749.56,A -85,B 0,C 180,E1 5900.262,E2 5900.262} C_VEL
LIN {X 0,Y 648.511,Z 749.56,A -85,B 0,C 180,E1 5905.992,E2 5905.992} C_VEL
LIN {X 0,Y 648.493,Z 749.56,A -85,B 0,C 180,E1 5910.697,E2 5910.697} C_VEL
LIN {X 0,Y 648.51,Z 749.56,A -85,B 0,C 180,E1 5915.336,E2 5915.336} C_VEL
LIN {X 0,Y 648.552,Z 749.56,A -85,B 0,C 180,E1 5920.957,E2 5920.957} C_VEL
LIN {X 0,Y 648.736,Z 749.56,A -85,B 0,C 180,E1 5926.526,E2 5926.526} C_VEL
LIN {X 0,Y 649.043,Z 749.56,A -85,B 0,C 180,E1 5931.966,E2 5931.966} C_VEL
LIN {X 0,Y 649.224,Z 749.56,A -85,B 0,C 180,E1 5937.328,E2 5937.328} C_VEL
LIN {X 0,Y 649.073,Z 749.56,A -85,B 0,C 180,E1 5942.665,E2 5942.665} C_VEL
LIN {X 0,Y 649.011,Z 749.56,A -85,B 0,C 180,E1 5946.682,E2 5946.682} C_VEL
LIN {X 0,Y 648.914,Z 749.56,A -85,B 0,C 180,E1 5952.094,E2 5952.094} C_VEL
LIN {X 0,Y 648.904,Z 749.56,A -85,B 0,C 180,E1 5957.619,E2 5957.619} C_VEL
LIN {X 0,Y 648.802,Z 749.56,A -85,B 0,C 180,E1 5961.876,E2 5961.876} C_VEL
LIN {X 0,Y 648.743,Z 749.56,A -85,B 0,C 180,E1 5966.265,E2 5966.265} C_VEL
LIN {X 0,Y 648.563,Z 749.56,A -85,B 0,C 180,E1 5971.687,E2 5971.687} C_VEL
LIN {X 0,Y 648.577,Z 749.56,A -85,B 0,C 180,E1 5974.687,E2 5974.687} C_VEL
LIN {X 0,Y 647.295,Z 749.56,A -85,B 0,C 180,E1 5975.453,E2 5975.453} C_VEL
LIN {X 0,Y 640.649,Z 749.56,A -85,B 0,C 180,E1 5977.533,E2 5977.533} C_VEL
LIN {X 0,Y 640.572,Z 749.56,A -85,B 0,C 180,E1 5977.73,E2 5977.73} C_VEL
LIN {X 0,Y 640.701,Z 749.56,A -85,B 0,C 180,E1 5983.152,E2 5983.152} C_VEL
LIN {X 0,Y 640.738,Z 750.184,A -85,B 0,C 180,E1 5984.943,E2 5984.943} C_VEL
LIN {X 0,Y 646.126,Z 760.44,A -85,B 0,C 180,E1 5985.554,E2 5985.554} C_VEL
LIN {X 0,Y 668.373,Z 799.121,A -85,B 0,C 180,E1 5987.947,E2 5987.947} C_VEL
LIN {X 0,Y 667.025,Z 855.12,A -85,B 0,C 180,E1 5988.839,E2 5988.839} C_VEL
LIN {X 0,Y 664.467,Z 898.565,A -85,B 0,C 180,E1 5989.973,E2 5989.973} C_VEL
LIN {X 0,Y 661.236,Z 945.203,A -85,B 0,C 180,E1 5991.749,E2 5991.749} C_VEL
LIN {X 0,Y 657.489,Z 989.799,A -85,B 0,C 180,E1 5994.017,E2 5994.017} C_VEL
LIN {X 0,Y 653.594,Z 1031.901,A -85,B 0,C 180,E1 5996.792,E2 5996.792} C_VEL
LIN {X 0,Y 649.94,Z 1070.846,A -85,B 0,C 180,E1 6000.007,E2 6000.007} C_VEL
LIN {X 0,Y 646.651,Z 1107.59,A -85,B 0,C 180,E1 6003.813,E2 6003.813} C_VEL
LIN {X 0,Y 644.375,Z 1137.437,A -85,B 0,C 180,E1 6007.692,E2 6007.692} C_VEL
LIN {X 0,Y 642.826,Z 1163.66,A -85,B 0,C 180,E1 6012.002,E2 6012.002} C_VEL
LIN {X 0,Y 641.904,Z 1183.702,A -85,B 0,C 180,E1 6016.383,E2 6016.383} C_VEL
LIN {X 0,Y 641.495,Z 1197.329,A -85,B 0,C 180,E1 6020.508,E2 6020.508} C_VEL
LIN {X 0,Y 641.338,Z 1205.909,A -85,B 0,C 180,E1 6024.591,E2 6024.591} C_VEL
LIN {X 0,Y 641.212,Z 1209.668,A -85,B 0,C 180,E1 6028.649,E2 6028.649} C_VEL
LIN {X 0,Y 641.393,Z 1208.939,A -85,B 0,C 180,E1 6032.7,E2 6032.7} C_VEL
LIN {X 0,Y 641.368,Z 1203.571,A -85,B 0,C 180,E1 6036.765,E2 6036.765} C_VEL
LIN {X 0,Y 641.571,Z 1192.317,A -85,B 0,C 180,E1 6041.204,E2 6041.204} C_VEL
LIN {X 0,Y 642.094,Z 1176.249,A -85,B 0,C 180,E1 6045.403,E2 6045.403} C_VEL
LIN {X 0,Y 643.147,Z 1155.807,A -85,B 0,C 180,E1 6049.412,E2 6049.412} C_VEL
LIN {X 0,Y 644.896,Z 1129.159,A -85,B 0,C 180,E1 6053.474,E2 6053.474} C_VEL
LIN {X 0,Y 647.613,Z 1096.568,A -85,B 0,C 180,E1 6057.428,E2 6057.428} C_VEL
LIN {X 0,Y 650.998,Z 1058.888,A -85,B 0,C 180,E1 6061.056,E2 6061.056} C_VEL
LIN {X 0,Y 654.685,Z 1020.408,A -85,B 0,C 180,E1 6064.036,E2 6064.036} C_VEL
LIN {X 0,Y 658.503,Z 978.158,A -85,B 0,C 180,E1 6066.629,E2 6066.629} C_VEL
LIN {X 0,Y 662.167,Z 933.935,A -85,B 0,C 180,E1 6068.738,E2 6068.738} C_VEL
LIN {X 0,Y 665.265,Z 886.115,A -85,B 0,C 180,E1 6070.396,E2 6070.396} C_VEL
LIN {X 0,Y 667.518,Z 839.333,A -85,B 0,C 180,E1 6071.473,E2 6071.473} C_VEL
LIN {X 0,Y 668.052,Z 798.766,A -85,B 0,C 180,E1 6072.083,E2 6072.083} C_VEL
LIN {X 0,Y 645.567,Z 759.511,A -85,B 0,C 180,E1 6074.509,E2 6074.509} C_VEL
LIN {X 0,Y 640.84,Z 750.891,A -85,B 0,C 180,E1 6075.036,E2 6075.036} C_VEL
LIN {X 0,Y 640.731,Z 749.56,A -85,B 0,C 180,E1 6075.083,E2 6075.083} C_VEL
LIN {X 0,Y 640.579,Z 749.56,A -85,B 0,C 180,E1 6081.12,E2 6081.12} C_VEL
LIN {X 0,Y 640.593,Z 749.56,A -85,B 0,C 180,E1 6085.652,E2 6085.652} C_VEL
LIN {X 0,Y 640.629,Z 749.56,A -85,B 0,C 180,E1 6090.78,E2 6090.78} C_VEL
LIN {X 0,Y 640.68,Z 749.56,A -85,B 0,C 180,E1 6094.881,E2 6094.881} C_VEL
LIN {X 0,Y 640.775,Z 749.56,A -85,B 0,C 180,E1 6100.725,E2 6100.725} C_VEL
LIN {X 0,Y 640.982,Z 749.56,A -85,B 0,C 180,E1 6105.144,E2 6105.144} C_VEL
LIN {X 0,Y 641.114,Z 749.56,A -85,B 0,C 180,E1 6110.507,E2 6110.507} C_VEL
LIN {X 0,Y 641.235,Z 749.56,A -85,B 0,C 180,E1 6115.95,E2 6115.95} C_VEL
LIN {X 0,Y 641.279,Z 749.56,A -85,B 0,C 180,E1 6120.004,E2 6120.004} C_VEL
LIN {X 0,Y 641.225,Z 749.56,A -85,B 0,C 180,E1 6124.058,E2 6124.058} C_VEL
LIN {X 0,Y 641.05,Z 749.56,A -85,B 0,C 180,E1 6129.502,E2 6129.502} C_VEL
LIN {X 0,Y 640.792,Z 749.56,A -85,B 0,C 180,E1 6135.039,E2 6135.039} C_VEL
LIN {X 0,Y 640.699,Z 749.56,A -85,B 0,C 180,E1 6140.723,E2 6140.723} C_VEL
LIN {X 0,Y 640.572,Z 749.56,A -85,B 0,C 180,E1 6146.634,E2 6146.634} C_VEL
LIN {X 0,Y 640.558,Z 749.56,A -85,B 0,C 180,E1 6151.869,E2 6151.869} C_VEL
LIN {X 0,Y 640.554,Z 749.56,A -85,B 0,C 180,E1 6156.671,E2 6156.671} C_VEL
LIN {X 0,Y 640.653,Z 750.263,A -85,B 0,C 180,E1 6160.994,E2 6160.994} C_VEL
LIN {X 0,Y 662.895,Z 793.744,A -85,B 0,C 180,E1 6163.399,E2 6163.399} C_VEL
LIN {X 0,Y 660.945,Z 839.408,A -85,B 0,C 180,E1 6164.478,E2 6164.478} C_VEL
LIN {X 0,Y 658.321,Z 882.33,A -85,B 0,C 180,E1 6166.012,E2 6166.012} C_VEL
LIN {X 0,Y 654.967,Z 925.918,A -85,B 0,C 180,E1 6168.124,E2 6168.124} C_VEL
LIN {X 0,Y 651.506,Z 967.637,A -85,B 0,C 180,E1 6170.811,E2 6170.811} C_VEL
LIN {X 0,Y 648.35,Z 1004.754,A -85,B 0,C 180,E1 6173.86,E2 6173.86} C_VEL
LIN {X 0,Y 645.643,Z 1039.155,A -85,B 0,C 180,E1 6177.432,E2 6177.432} C_VEL
LIN {X 0,Y 643.632,Z 1067.974,A -85,B 0,C 180,E1 6181.252,E2 6181.252} C_VEL
LIN {X 0,Y 642.414,Z 1089.813,A -85,B 0,C 180,E1 6184.951,E2 6184.951} C_VEL
LIN {X 0,Y 641.747,Z 1107.109,A -85,B 0,C 180,E1 6188.812,E2 6188.812} C_VEL
LIN {X 0,Y 641.37,Z 1118.971,A -85,B 0,C 180,E1 6192.489,E2 6192.489} C_VEL
LIN {X 0,Y 641.248,Z 1126.726,A -85,B 0,C 180,E1 6196.371,E2 6196.371} C_VEL
LIN {X 0,Y 641.221,Z 1129.895,A -85,B 0,C 180,E1 6200.505,E2 6200.505} C_VEL
LIN {X 0,Y 641.287,Z 1127.923,A -85,B 0,C 180,E1 6204.592,E2 6204.592} C_VEL
LIN {X 0,Y 641.344,Z 1120.835,A -85,B 0,C 180,E1 6208.651,E2 6208.651} C_VEL
LIN {X 0,Y 641.632,Z 1109.888,A -85,B 0,C 180,E1 6212.363,E2 6212.363} C_VEL
LIN {X 0,Y 642.16,Z 1094.229,A -85,B 0,C 180,E1 6216.079,E2 6216.079} C_VEL
LIN {X 0,Y 643.436,Z 1071.363,A -85,B 0,C 180,E1 6220.146,E2 6220.146} C_VEL
LIN {X 0,Y 645.162,Z 1044.017,A -85,B 0,C 180,E1 6223.892,E2 6223.892} C_VEL
LIN {X 0,Y 647.808,Z 1011.79,A -85,B 0,C 180,E1 6227.387,E2 6227.387} C_VEL
LIN {X 0,Y 651.124,Z 972.729,A -85,B 0,C 180,E1 6230.728,E2 6230.728} C_VEL
LIN {X 0,Y 654.663,Z 929.982,A -85,B 0,C 180,E1 6233.549,E2 6233.549} C_VEL
LIN {X 0,Y 657.902,Z 887.247,A -85,B 0,C 180,E1 6235.693,E2 6235.693} C_VEL
LIN {X 0,Y 660.87,Z 842.193,A -85,B 0,C 180,E1 6237.347,E2 6237.347} C_VEL
LIN {X 0,Y 662.83,Z 800.909,A -85,B 0,C 180,E1 6238.365,E2 6238.365} C_VEL
LIN {X 0,Y 662.202,Z 792.591,A -85,B 0,C 180,E1 6238.581,E2 6238.581} C_VEL
LIN {X 0,Y 642.821,Z 754.905,A -85,B 0,C 180,E1 6240.649,E2 6240.649} C_VEL
LIN {X 0,Y 640.694,Z 749.56,A -85,B 0,C 180,E1 6240.906,E2 6240.906} C_VEL
LIN {X 0,Y 640.596,Z 749.56,A -85,B 0,C 180,E1 6246.139,E2 6246.139} C_VEL
LIN {X 0,Y 640.645,Z 749.56,A -85,B 0,C 180,E1 6251.335,E2 6251.335} C_VEL
LIN {X 0,Y 640.604,Z 749.56,A -85,B 0,C 180,E1 6256.83,E2 6256.83} C_VEL
LIN {X 0,Y 640.588,Z 749.56,A -85,B 0,C 180,E1 6262.163,E2 6262.163} C_VEL
LIN {X 0,Y 640.587,Z 749.56,A -85,B 0,C 180,E1 6267.136,E2 6267.136} C_VEL
LIN {X 0,Y 640.562,Z 749.56,A -85,B 0,C 180,E1 6271.843,E2 6271.843} C_VEL
LIN {X 0,Y 640.57,Z 749.56,A -85,B 0,C 180,E1 6276.931,E2 6276.931} C_VEL
LIN {X 0,Y 640.606,Z 749.56,A -85,B 0,C 180,E1 6282.138,E2 6282.138} C_VEL
LIN {X 0,Y 640.814,Z 749.56,A -85,B 0,C 180,E1 6286.356,E2 6286.356} C_VEL
LIN {X 0,Y 641.061,Z 749.56,A -85,B 0,C 180,E1 6290.498,E2 6290.498} C_VEL
LIN {X 0,Y 641.22,Z 749.56,A -85,B 0,C 180,E1 6295.942,E2 6295.942} C_VEL
LIN {X 0,Y 641.434,Z 749.56,A -85,B 0,C 180,E1 6301.346,E2 6301.346} C_VEL
LIN {X 0,Y 641.102,Z 749.56,A -85,B 0,C 180,E1 6306.765,E2 6306.765} C_VEL
LIN {X 0,Y 640.993,Z 749.56,A -85,B 0,C 180,E1 6312.246,E2 6312.246} C_VEL
LIN {X 0,Y 640.973,Z 749.56,A -85,B 0,C 180,E1 6317.844,E2 6317.844} C_VEL
LIN {X 0,Y 640.864,Z 749.56,A -85,B 0,C 180,E1 6323.13,E2 6323.13} C_VEL
LIN {X 0,Y 640.767,Z 749.56,A -85,B 0,C 180,E1 6328.139,E2 6328.139} C_VEL
LIN {X 0,Y 640.712,Z 749.56,A -85,B 0,C 180,E1 6332.848,E2 6332.848} C_VEL
LIN {X 0,Y 640.572,Z 749.56,A -85,B 0,C 180,E1 6337.73,E2 6337.73} C_VEL
LIN {X 0,Y 638.087,Z 749.56,A -85,B 0,C 180,E1 6338.874,E2 6338.874} C_VEL
LIN {X 0,Y 632.697,Z 749.56,A -85,B 0,C 180,E1 6340.584,E2 6340.584} C_VEL
LIN {X 0,Y 632.598,Z 749.56,A -85,B 0,C 180,E1 6340.782,E2 6340.782} C_VEL
LIN {X 0,Y 632.849,Z 750.127,A -85,B 0,C 180,E1 6344.289,E2 6344.289} C_VEL
LIN {X 0,Y 641.321,Z 765.541,A -85,B 0,C 180,E1 6345.217,E2 6345.217} C_VEL
LIN {X 0,Y 662.327,Z 801.742,A -85,B 0,C 180,E1 6347.511,E2 6347.511} C_VEL
LIN {X 0,Y 660.954,Z 857.312,A -85,B 0,C 180,E1 6348.434,E2 6348.434} C_VEL
LIN {X 0,Y 658.13,Z 901.234,A -85,B 0,C 180,E1 6349.611,E2 6349.611} C_VEL
LIN {X 0,Y 654.511,Z 949.809,A -85,B 0,C 180,E1 6351.513,E2 6351.513} C_VEL
LIN {X 0,Y 650.328,Z 994.806,A -85,B 0,C 180,E1 6353.895,E2 6353.895} C_VEL
LIN {X 0,Y 646.061,Z 1038.57,A -85,B 0,C 180,E1 6356.889,E2 6356.889} C_VEL
LIN {X 0,Y 642.006,Z 1078.513,A -85,B 0,C 180,E1 6360.376,E2 6360.376} C_VEL
LIN {X 0,Y 638.846,Z 1111.908,A -85,B 0,C 180,E1 6364.002,E2 6364.002} C_VEL
LIN {X 0,Y 636.295,Z 1143.264,A -85,B 0,C 180,E1 6368.281,E2 6368.281} C_VEL
LIN {X 0,Y 634.858,Z 1167.17,A -85,B 0,C 180,E1 6372.473,E2 6372.473} C_VEL
LIN {X 0,Y 633.893,Z 1186.378,A -85,B 0,C 180,E1 6376.91,E2 6376.91} C_VEL
LIN {X 0,Y 633.513,Z 1199.101,A -85,B 0,C 180,E1 6381.08,E2 6381.08} C_VEL
LIN {X 0,Y 633.441,Z 1205.909,A -85,B 0,C 180,E1 6384.524,E2 6384.524} C_VEL
LIN {X 0,Y 633.331,Z 1209.667,A -85,B 0,C 180,E1 6388.632,E2 6388.632} C_VEL
LIN {X 0,Y 633.501,Z 1208.936,A -85,B 0,C 180,E1 6392.734,E2 6392.734} C_VEL
LIN {X 0,Y 633.472,Z 1203.571,A -85,B 0,C 180,E1 6396.849,E2 6396.849} C_VEL
LIN {X 0,Y 633.69,Z 1193.42,A -85,B 0,C 180,E1 6400.997,E2 6400.997} C_VEL
LIN {X 0,Y 634.25,Z 1177.036,A -85,B 0,C 180,E1 6405.419,E2 6405.419} C_VEL
LIN {X 0,Y 635.329,Z 1156.962,A -85,B 0,C 180,E1 6409.45,E2 6409.45} C_VEL
LIN {X 0,Y 637.145,Z 1131.803,A -85,B 0,C 180,E1 6413.406,E2 6413.406} C_VEL
LIN {X 0,Y 640.033,Z 1098.975,A -85,B 0,C 180,E1 6417.498,E2 6417.498} C_VEL
LIN {X 0,Y 643.534,Z 1062.657,A -85,B 0,C 180,E1 6421.104,E2 6421.104} C_VEL
LIN {X 0,Y 647.714,Z 1022.076,A -85,B 0,C 180,E1 6424.33,E2 6424.33} C_VEL
LIN {X 0,Y 651.86,Z 979.542,A -85,B 0,C 180,E1 6426.98,E2 6426.98} C_VEL
LIN {X 0,Y 655.829,Z 934.615,A -85,B 0,C 180,E1 6429.15,E2 6429.15} C_VEL
LIN {X 0,Y 659.051,Z 888.022,A -85,B 0,C 180,E1 6430.793,E2 6430.793} C_VEL
LIN {X 0,Y 661.487,Z 841.25,A -85,B 0,C 180,E1 6431.893,E2 6431.893} C_VEL
LIN {X 0,Y 662.019,Z 801.638,A -85,B 0,C 180,E1 6432.515,E2 6432.515} C_VEL
LIN {X 0,Y 638.43,Z 760.795,A -85,B 0,C 180,E1 6435.084,E2 6435.084} C_VEL
LIN {X 0,Y 632.946,Z 751.065,A -85,B 0,C 180,E1 6435.676,E2 6435.676} C_VEL
LIN {X 0,Y 632.78,Z 749.56,A -85,B 0,C 180,E1 6435.759,E2 6435.759} C_VEL
LIN {X 0,Y 632.668,Z 749.56,A -85,B 0,C 180,E1 6441.614,E2 6441.614} C_VEL
LIN {X 0,Y 632.647,Z 749.56,A -85,B 0,C 180,E1 6446.719,E2 6446.719} C_VEL
LIN {X 0,Y 632.68,Z 749.56,A -85,B 0,C 180,E1 6452.094,E2 6452.094} C_VEL
LIN {X 0,Y 632.762,Z 749.56,A -85,B 0,C 180,E1 6457.539,E2 6457.539} C_VEL
LIN {X 0,Y 632.983,Z 749.56,A -85,B 0,C 180,E1 6462.729,E2 6462.729} C_VEL
LIN {X 0,Y 633.086,Z 749.56,A -85,B 0,C 180,E1 6468.132,E2 6468.132} C_VEL
LIN {X 0,Y 633.188,Z 749.56,A -85,B 0,C 180,E1 6473.15,E2 6473.15} C_VEL
LIN {X 0,Y 633.518,Z 749.56,A -85,B 0,C 180,E1 6478.637,E2 6478.637} C_VEL
LIN {X 0,Y 633.324,Z 749.56,A -85,B 0,C 180,E1 6484.109,E2 6484.109} C_VEL
LIN {X 0,Y 633.134,Z 749.56,A -85,B 0,C 180,E1 6489.622,E2 6489.622} C_VEL
LIN {X 0,Y 632.851,Z 749.56,A -85,B 0,C 180,E1 6495.232,E2 6495.232} C_VEL
LIN {X 0,Y 632.753,Z 749.56,A -85,B 0,C 180,E1 6500.996,E2 6500.996} C_VEL
LIN {X 0,Y 632.644,Z 749.56,A -85,B 0,C 180,E1 6505.469,E2 6505.469} C_VEL
LIN {X 0,Y 632.642,Z 749.56,A -85,B 0,C 180,E1 6510.696,E2 6510.696} C_VEL
LIN {X 0,Y 632.631,Z 749.56,A -85,B 0,C 180,E1 6515.696,E2 6515.696} C_VEL
LIN {X 0,Y 632.682,Z 749.56,A -85,B 0,C 180,E1 6520.293,E2 6520.293} C_VEL
LIN {X 0,Y 635.26,Z 755.356,A -85,B 0,C 180,E1 6520.617,E2 6520.617} C_VEL
LIN {X 0,Y 654.947,Z 793.146,A -85,B 0,C 180,E1 6522.844,E2 6522.844} C_VEL
LIN {X 0,Y 656.575,Z 798.626,A -85,B 0,C 180,E1 6523.078,E2 6523.078} C_VEL
LIN {X 0,Y 654.467,Z 841.115,A -85,B 0,C 180,E1 6524.112,E2 6524.112} C_VEL
LIN {X 0,Y 651.454,Z 886.013,A -85,B 0,C 180,E1 6525.764,E2 6525.764} C_VEL
LIN {X 0,Y 647.945,Z 928.15,A -85,B 0,C 180,E1 6527.863,E2 6527.863} C_VEL
LIN {X 0,Y 644.144,Z 971.109,A -85,B 0,C 180,E1 6530.699,E2 6530.699} C_VEL
LIN {X 0,Y 640.73,Z 1008.393,A -85,B 0,C 180,E1 6533.871,E2 6533.871} C_VEL
LIN {X 0,Y 638.04,Z 1039.906,A -85,B 0,C 180,E1 6537.229,E2 6537.229} C_VEL
LIN {X 0,Y 635.826,Z 1069.778,A -85,B 0,C 180,E1 6541.272,E2 6541.272} C_VEL
LIN {X 0,Y 634.529,Z 1091.731,A -85,B 0,C 180,E1 6545.135,E2 6545.135} C_VEL
LIN {X 0,Y 633.827,Z 1108.594,A -85,B 0,C 180,E1 6549.047,E2 6549.047} C_VEL
LIN {X 0,Y 633.458,Z 1119.585,A -85,B 0,C 180,E1 6552.611,E2 6552.611} C_VEL
LIN {X 0,Y 633.363,Z 1126.581,A -85,B 0,C 180,E1 6556.197,E2 6556.197} C_VEL
LIN {X 0,Y 633.297,Z 1129.867,A -85,B 0,C 180,E1 6560.386,E2 6560.386} C_VEL
LIN {X 0,Y 633.379,Z 1128.064,A -85,B 0,C 180,E1 6564.524,E2 6564.524} C_VEL
LIN {X 0,Y 633.478,Z 1122.641,A -85,B 0,C 180,E1 6567.95,E2 6567.95} C_VEL
LIN {X 0,Y 633.678,Z 1112.53,A -85,B 0,C 180,E1 6571.709,E2 6571.709} C_VEL
LIN {X 0,Y 634.272,Z 1096.44,A -85,B 0,C 180,E1 6575.812,E2 6575.812} C_VEL
LIN {X 0,Y 635.394,Z 1075.254,A -85,B 0,C 180,E1 6579.757,E2 6579.757} C_VEL
LIN {X 0,Y 637.165,Z 1049.686,A -85,B 0,C 180,E1 6583.477,E2 6583.477} C_VEL
LIN {X 0,Y 640.06,Z 1016.626,A -85,B 0,C 180,E1 6587.232,E2 6587.232} C_VEL
LIN {X 0,Y 643.149,Z 981.839,A -85,B 0,C 180,E1 6590.369,E2 6590.369} C_VEL
LIN {X 0,Y 646.777,Z 942.883,A -85,B 0,C 180,E1 6593.157,E2 6593.157} C_VEL
LIN {X 0,Y 650.29,Z 901.025,A -85,B 0,C 180,E1 6595.462,E2 6595.462} C_VEL
LIN {X 0,Y 653.451,Z 858.639,A -85,B 0,C 180,E1 6597.221,E2 6597.221} C_VEL
LIN {X 0,Y 655.908,Z 812.525,A -85,B 0,C 180,E1 6598.547,E2 6598.547} C_VEL
LIN {X 0,Y 656.098,Z 796.063,A -85,B 0,C 180,E1 6598.919,E2 6598.919} C_VEL
LIN {X 0,Y 638.38,Z 760.719,A -85,B 0,C 180,E1 6600.925,E2 6600.925} C_VEL
LIN {X 0,Y 632.936,Z 751.344,A -85,B 0,C 180,E1 6601.521,E2 6601.521} C_VEL
LIN {X 0,Y 632.744,Z 749.56,A -85,B 0,C 180,E1 6601.614,E2 6601.614} C_VEL
LIN {X 0,Y 632.693,Z 749.56,A -85,B 0,C 180,E1 6606.663,E2 6606.663} C_VEL
LIN {X 0,Y 632.714,Z 749.56,A -85,B 0,C 180,E1 6612.229,E2 6612.229} C_VEL
LIN {X 0,Y 632.633,Z 749.56,A -85,B 0,C 180,E1 6618.018,E2 6618.018} C_VEL
LIN {X 0,Y 632.673,Z 749.56,A -85,B 0,C 180,E1 6623.33,E2 6623.33} C_VEL
LIN {X 0,Y 632.64,Z 749.56,A -85,B 0,C 180,E1 6628.293,E2 6628.293} C_VEL
LIN {X 0,Y 632.639,Z 749.56,A -85,B 0,C 180,E1 6633.005,E2 6633.005} C_VEL
LIN {X 0,Y 632.684,Z 749.56,A -85,B 0,C 180,E1 6638.67,E2 6638.67} C_VEL
LIN {X 0,Y 632.73,Z 749.56,A -85,B 0,C 180,E1 6643.342,E2 6643.342} C_VEL
LIN {X 0,Y 633.117,Z 749.56,A -85,B 0,C 180,E1 6648.988,E2 6648.988} C_VEL
LIN {X 0,Y 633.216,Z 749.56,A -85,B 0,C 180,E1 6654.518,E2 6654.518} C_VEL
LIN {X 0,Y 633.308,Z 749.56,A -85,B 0,C 180,E1 6658.629,E2 6658.629} C_VEL
LIN {X 0,Y 633.279,Z 749.56,A -85,B 0,C 180,E1 6662.732,E2 6662.732} C_VEL
LIN {X 0,Y 633.195,Z 749.56,A -85,B 0,C 180,E1 6666.85,E2 6666.85} C_VEL
LIN {X 0,Y 633.09,Z 749.56,A -85,B 0,C 180,E1 6672.401,E2 6672.401} C_VEL
LIN {X 0,Y 633.057,Z 749.56,A -85,B 0,C 180,E1 6678.075,E2 6678.075} C_VEL
LIN {X 0,Y 632.942,Z 749.56,A -85,B 0,C 180,E1 6682.454,E2 6682.454} C_VEL
LIN {X 0,Y 632.878,Z 749.56,A -85,B 0,C 180,E1 6687.937,E2 6687.937} C_VEL
LIN {X 0,Y 632.772,Z 749.56,A -85,B 0,C 180,E1 6693.313,E2 6693.313} C_VEL
LIN {X 0,Y 632.662,Z 749.56,A -85,B 0,C 180,E1 6698.387,E2 6698.387} C_VEL
LIN {X 0,Y 632.598,Z 749.56,A -85,B 0,C 180,E1 6700.782,E2 6700.782} C_VEL
LIN {X 0,Y 628.694,Z 749.56,A -85,B 0,C 180,E1 6701.794,E2 6701.794} C_VEL
LIN {X 0,Y 624.791,Z 749.56,A -85,B 0,C 180,E1 6702.818,E2 6702.818} C_VEL
LIN {X 0,Y 624.877,Z 749.959,A -85,B 0,C 180,E1 6703.603,E2 6703.603} C_VEL
LIN {X 0,Y 627.694,Z 755.595,A -85,B 0,C 180,E1 6703.934,E2 6703.934} C_VEL
LIN {X 0,Y 656.395,Z 804.969,A -85,B 0,C 180,E1 6707.082,E2 6707.082} C_VEL
LIN {X 0,Y 654.949,Z 858.584,A -85,B 0,C 180,E1 6708.001,E2 6708.001} C_VEL
LIN {X 0,Y 651.891,Z 903.198,A -85,B 0,C 180,E1 6709.221,E2 6709.221} C_VEL
LIN {X 0,Y 648.033,Z 951.726,A -85,B 0,C 180,E1 6711.153,E2 6711.153} C_VEL
LIN {X 0,Y 643.61,Z 996.159,A -85,B 0,C 180,E1 6713.551,E2 6713.551} C_VEL
LIN {X 0,Y 639.106,Z 1039.005,A -85,B 0,C 180,E1 6716.519,E2 6716.519} C_VEL
LIN {X 0,Y 634.692,Z 1079.604,A -85,B 0,C 180,E1 6720.112,E2 6720.112} C_VEL
LIN {X 0,Y 631.318,Z 1112.908,A -85,B 0,C 180,E1 6723.798,E2 6723.798} C_VEL
LIN {X 0,Y 628.63,Z 1143.728,A -85,B 0,C 180,E1 6728.075,E2 6728.075} C_VEL
LIN {X 0,Y 627.078,Z 1167.566,A -85,B 0,C 180,E1 6732.33,E2 6732.33} C_VEL
LIN {X 0,Y 626.067,Z 1186.377,A -85,B 0,C 180,E1 6736.743,E2 6736.743} C_VEL
LIN {X 0,Y 625.638,Z 1199.102,A -85,B 0,C 180,E1 6740.967,E2 6740.967} C_VEL
LIN {X 0,Y 625.546,Z 1205.909,A -85,B 0,C 180,E1 6744.454,E2 6744.454} C_VEL
LIN {X 0,Y 625.431,Z 1209.667,A -85,B 0,C 180,E1 6748.615,E2 6748.615} C_VEL
LIN {X 0,Y 625.593,Z 1208.933,A -85,B 0,C 180,E1 6752.768,E2 6752.768} C_VEL
LIN {X 0,Y 625.577,Z 1203.571,A -85,B 0,C 180,E1 6756.936,E2 6756.936} C_VEL
LIN {X 0,Y 625.822,Z 1193.421,A -85,B 0,C 180,E1 6761.137,E2 6761.137} C_VEL
LIN {X 0,Y 626.384,Z 1178.012,A -85,B 0,C 180,E1 6765.388,E2 6765.388} C_VEL
LIN {X 0,Y 627.467,Z 1158.938,A -85,B 0,C 180,E1 6769.337,E2 6769.337} C_VEL
LIN {X 0,Y 629.476,Z 1133.124,A -85,B 0,C 180,E1 6773.521,E2 6773.521} C_VEL
LIN {X 0,Y 632.502,Z 1100.821,A -85,B 0,C 180,E1 6777.632,E2 6777.632} C_VEL
LIN {X 0,Y 636.15,Z 1065.57,A -85,B 0,C 180,E1 6781.228,E2 6781.228} C_VEL
LIN {X 0,Y 640.642,Z 1024.609,A -85,B 0,C 180,E1 6784.56,E2 6784.56} C_VEL
LIN {X 0,Y 644.936,Z 983.577,A -85,B 0,C 180,E1 6787.194,E2 6787.194} C_VEL
LIN {X 0,Y 649.211,Z 938.371,A -85,B 0,C 180,E1 6789.437,E2 6789.437} C_VEL
LIN {X 0,Y 652.759,Z 892.315,A -85,B 0,C 180,E1 6791.127,E2 6791.127} C_VEL
LIN {X 0,Y 655.487,Z 843.475,A -85,B 0,C 180,E1 6792.314,E2 6792.314} C_VEL
LIN {X 0,Y 656.072,Z 804.705,A -85,B 0,C 180,E1 6792.948,E2 6792.948} C_VEL
LIN {X 0,Y 633.806,Z 766.351,A -85,B 0,C 180,E1 6795.376,E2 6795.376} C_VEL
LIN {X 0,Y 624.855,Z 750.491,A -85,B 0,C 180,E1 6796.368,E2 6796.368} C_VEL
LIN {X 0,Y 624.772,Z 749.56,A -85,B 0,C 180,E1 6796.518,E2 6796.518} C_VEL
LIN {X 0,Y 624.702,Z 749.56,A -85,B 0,C 180,E1 6801.033,E2 6801.033} C_VEL
LIN {X 0,Y 624.686,Z 749.56,A -85,B 0,C 180,E1 6806.198,E2 6806.198} C_VEL
LIN {X 0,Y 624.737,Z 749.56,A -85,B 0,C 180,E1 6811.072,E2 6811.072} C_VEL
LIN {X 0,Y 624.844,Z 749.56,A -85,B 0,C 180,E1 6815.728,E2 6815.728} C_VEL
LIN {X 0,Y 624.994,Z 749.56,A -85,B 0,C 180,E1 6820.551,E2 6820.551} C_VEL
LIN {X 0,Y 625.152,Z 749.56,A -85,B 0,C 180,E1 6826.015,E2 6826.015} C_VEL
LIN {X 0,Y 625.308,Z 749.56,A -85,B 0,C 180,E1 6831.667,E2 6831.667} C_VEL
LIN {X 0,Y 625.431,Z 749.56,A -85,B 0,C 180,E1 6835.847,E2 6835.847} C_VEL
LIN {X 0,Y 625.506,Z 749.56,A -85,B 0,C 180,E1 6840.004,E2 6840.004} C_VEL
LIN {X 0,Y 625.413,Z 749.56,A -85,B 0,C 180,E1 6844.161,E2 6844.161} C_VEL
LIN {X 0,Y 625.233,Z 749.56,A -85,B 0,C 180,E1 6849.744,E2 6849.744} C_VEL
LIN {X 0,Y 624.936,Z 749.56,A -85,B 0,C 180,E1 6855.43,E2 6855.43} C_VEL
LIN {X 0,Y 624.852,Z 749.56,A -85,B 0,C 180,E1 6861.274,E2 6861.274} C_VEL
LIN {X 0,Y 624.685,Z 749.56,A -85,B 0,C 180,E1 6866.488,E2 6866.488} C_VEL
LIN {X 0,Y 624.721,Z 749.56,A -85,B 0,C 180,E1 6872.157,E2 6872.157} C_VEL
LIN {X 0,Y 624.743,Z 749.56,A -85,B 0,C 180,E1 6877.213,E2 6877.213} C_VEL
LIN {X 0,Y 624.751,Z 749.802,A -85,B 0,C 180,E1 6879.613,E2 6879.613} C_VEL
LIN {X 0,Y 627.143,Z 755.222,A -85,B 0,C 180,E1 6879.91,E2 6879.91} C_VEL
LIN {X 0,Y 644.416,Z 786.694,A -85,B 0,C 180,E1 6881.887,E2 6881.887} C_VEL
LIN {X 0,Y 650.42,Z 800.301,A -85,B 0,C 180,E1 6882.664,E2 6882.664} C_VEL
LIN {X 0,Y 648.002,Z 842.914,A -85,B 0,C 180,E1 6883.747,E2 6883.747} C_VEL
LIN {X 0,Y 644.795,Z 887.21,A -85,B 0,C 180,E1 6885.403,E2 6885.403} C_VEL
LIN {X 0,Y 641.142,Z 928.475,A -85,B 0,C 180,E1 6887.487,E2 6887.487} C_VEL
LIN {X 0,Y 637.052,Z 971.701,A -85,B 0,C 180,E1 6890.373,E2 6890.373} C_VEL
LIN {X 0,Y 633.327,Z 1009.632,A -85,B 0,C 180,E1 6893.653,E2 6893.653} C_VEL
LIN {X 0,Y 630.375,Z 1041.505,A -85,B 0,C 180,E1 6897.126,E2 6897.126} C_VEL
LIN {X 0,Y 628.112,Z 1070.114,A -85,B 0,C 180,E1 6901.071,E2 6901.071} C_VEL
LIN {X 0,Y 626.656,Z 1092.911,A -85,B 0,C 180,E1 6905.175,E2 6905.175} C_VEL
LIN {X 0,Y 625.944,Z 1109.506,A -85,B 0,C 180,E1 6909.141,E2 6909.141} C_VEL
LIN {X 0,Y 625.501,Z 1121.026,A -85,B 0,C 180,E1 6913.149,E2 6913.149} C_VEL
LIN {X 0,Y 625.465,Z 1126.435,A -85,B 0,C 180,E1 6916.02,E2 6916.02} C_VEL
LIN {X 0,Y 625.404,Z 1129.839,A -85,B 0,C 180,E1 6920.263,E2 6920.263} C_VEL
LIN {X 0,Y 625.471,Z 1128.205,A -85,B 0,C 180,E1 6924.455,E2 6924.455} C_VEL
LIN {X 0,Y 625.603,Z 1122.898,A -85,B 0,C 180,E1 6927.924,E2 6927.924} C_VEL
LIN {X 0,Y 625.801,Z 1111.78,A -85,B 0,C 180,E1 6932.076,E2 6932.076} C_VEL
LIN {X 0,Y 626.427,Z 1096.949,A -85,B 0,C 180,E1 6935.885,E2 6935.885} C_VEL
LIN {X 0,Y 627.655,Z 1075.961,A -85,B 0,C 180,E1 6939.878,E2 6939.878} C_VEL
LIN {X 0,Y 629.701,Z 1048.705,A -85,B 0,C 180,E1 6943.886,E2 6943.886} C_VEL
LIN {X 0,Y 632.881,Z 1014.79,A -85,B 0,C 180,E1 6947.754,E2 6947.754} C_VEL
LIN {X 0,Y 636.526,Z 976.809,A -85,B 0,C 180,E1 6951.135,E2 6951.135} C_VEL
LIN {X 0,Y 640.324,Z 937.553,A -85,B 0,C 180,E1 6953.874,E2 6953.874} C_VEL
LIN {X 0,Y 644.199,Z 894.511,A -85,B 0,C 180,E1 6956.187,E2 6956.187} C_VEL
LIN {X 0,Y 647.474,Z 851.393,A -85,B 0,C 180,E1 6957.881,E2 6957.881} C_VEL
LIN {X 0,Y 650.037,Z 808.455,A -85,B 0,C 180,E1 6959.074,E2 6959.074} C_VEL
LIN {X 0,Y 649.875,Z 798.933,A -85,B 0,C 180,E1 6959.314,E2 6959.314} C_VEL
LIN {X 0,Y 633.146,Z 765.369,A -85,B 0,C 180,E1 6961.29,E2 6961.29} C_VEL
LIN {X 0,Y 624.91,Z 750.992,A -85,B 0,C 180,E1 6962.219,E2 6962.219} C_VEL
LIN {X 0,Y 624.777,Z 749.56,A -85,B 0,C 180,E1 6962.348,E2 6962.348} C_VEL
LIN {X 0,Y 624.758,Z 749.56,A -85,B 0,C 180,E1 6967.207,E2 6967.207} C_VEL
LIN {X 0,Y 624.796,Z 749.56,A -85,B 0,C 180,E1 6972.627,E2 6972.627} C_VEL
LIN {X 0,Y 624.716,Z 749.56,A -85,B 0,C 180,E1 6977.361,E2 6977.361} C_VEL
LIN {X 0,Y 624.756,Z 749.56,A -85,B 0,C 180,E1 6982.958,E2 6982.958} C_VEL
LIN {X 0,Y 624.701,Z 749.56,A -85,B 0,C 180,E1 6987.849,E2 6987.849} C_VEL
LIN {X 0,Y 624.696,Z 749.56,A -85,B 0,C 180,E1 6993.513,E2 6993.513} C_VEL
LIN {X 0,Y 624.817,Z 749.56,A -85,B 0,C 180,E1 6998.725,E2 6998.725} C_VEL
LIN {X 0,Y 624.939,Z 749.56,A -85,B 0,C 180,E1 7004.57,E2 7004.57} C_VEL
LIN {X 0,Y 625.243,Z 749.56,A -85,B 0,C 180,E1 7010.256,E2 7010.256} C_VEL
LIN {X 0,Y 625.41,Z 749.56,A -85,B 0,C 180,E1 7015.839,E2 7015.839} C_VEL
LIN {X 0,Y 625.63,Z 749.56,A -85,B 0,C 180,E1 7021.38,E2 7021.38} C_VEL
LIN {X 0,Y 625.285,Z 749.56,A -85,B 0,C 180,E1 7026.937,E2 7026.937} C_VEL
LIN {X 0,Y 625.17,Z 749.56,A -85,B 0,C 180,E1 7032.561,E2 7032.561} C_VEL
LIN {X 0,Y 625.171,Z 749.56,A -85,B 0,C 180,E1 7036.858,E2 7036.858} C_VEL
LIN {X 0,Y 625.074,Z 749.56,A -85,B 0,C 180,E1 7041.258,E2 7041.258} C_VEL
LIN {X 0,Y 624.928,Z 749.56,A -85,B 0,C 180,E1 7046.53,E2 7046.53} C_VEL
LIN {X 0,Y 624.862,Z 749.56,A -85,B 0,C 180,E1 7052.175,E2 7052.175} C_VEL
LIN {X 0,Y 624.775,Z 749.56,A -85,B 0,C 180,E1 7057.201,E2 7057.201} C_VEL
LIN {X 0,Y 624.791,Z 749.56,A -85,B 0,C 180,E1 7062.818,E2 7062.818} C_VEL
LIN {X 0,Y 625.404,Z 753.082,A -85,B 0,C 180,E1 7063.48,E2 7063.48} C_VEL
LIN {X 0,Y 627.949,Z 764.625,A -85,B 0,C 180,E1 7064.094,E2 7064.094} C_VEL
LIN {X 0,Y 632.48,Z 777.088,A -85,B 0,C 180,E1 7064.666,E2 7064.666} C_VEL
LIN {X 0,Y 650.687,Z 808.385,A -85,B 0,C 180,E1 7066.664,E2 7066.664} C_VEL
LIN {X 0,Y 648.96,Z 860.03,A -85,B 0,C 180,E1 7067.566,E2 7067.566} C_VEL
LIN {X 0,Y 645.659,Z 905.319,A -85,B 0,C 180,E1 7068.826,E2 7068.826} C_VEL
LIN {X 0,Y 641.674,Z 952.475,A -85,B 0,C 180,E1 7070.735,E2 7070.735} C_VEL
LIN {X 0,Y 636.791,Z 998.433,A -85,B 0,C 180,E1 7073.254,E2 7073.254} C_VEL
LIN {X 0,Y 632.154,Z 1039.808,A -85,B 0,C 180,E1 7076.173,E2 7076.173} C_VEL
LIN {X 0,Y 627.441,Z 1080.243,A -85,B 0,C 180,E1 7079.798,E2 7079.798} C_VEL
LIN {X 0,Y 623.864,Z 1113.358,A -85,B 0,C 180,E1 7083.519,E2 7083.519} C_VEL
LIN {X 0,Y 621.003,Z 1143.963,A -85,B 0,C 180,E1 7087.829,E2 7087.829} C_VEL
LIN {X 0,Y 619.262,Z 1168.074,A -85,B 0,C 180,E1 7092.205,E2 7092.205} C_VEL
LIN {X 0,Y 618.251,Z 1186.376,A -85,B 0,C 180,E1 7096.573,E2 7096.573} C_VEL
LIN {X 0,Y 617.774,Z 1199.102,A -85,B 0,C 180,E1 7100.851,E2 7100.851} C_VEL
LIN {X 0,Y 617.652,Z 1205.909,A -85,B 0,C 180,E1 7104.383,E2 7104.383} C_VEL
LIN {X 0,Y 617.547,Z 1209.667,A -85,B 0,C 180,E1 7108.597,E2 7108.597} C_VEL
LIN {X 0,Y 617.708,Z 1208.931,A -85,B 0,C 180,E1 7112.804,E2 7112.804} C_VEL
LIN {X 0,Y 617.705,Z 1203.571,A -85,B 0,C 180,E1 7117.025,E2 7117.025} C_VEL
LIN {X 0,Y 617.931,Z 1193.421,A -85,B 0,C 180,E1 7121.281,E2 7121.281} C_VEL
LIN {X 0,Y 618.564,Z 1178.011,A -85,B 0,C 180,E1 7125.588,E2 7125.588} C_VEL
LIN {X 0,Y 619.754,Z 1158.94,A -85,B 0,C 180,E1 7129.588,E2 7129.588} C_VEL
LIN {X 0,Y 621.886,Z 1133.122,A -85,B 0,C 180,E1 7133.826,E2 7133.826} C_VEL
LIN {X 0,Y 625.136,Z 1101.109,A -85,B 0,C 180,E1 7137.952,E2 7137.952} C_VEL
LIN {X 0,Y 629.112,Z 1065.57,A -85,B 0,C 180,E1 7141.618,E2 7141.618} C_VEL
LIN {X 0,Y 633.966,Z 1023.699,A -85,B 0,C 180,E1 7145.052,E2 7145.052} C_VEL
LIN {X 0,Y 638.645,Z 982.22,A -85,B 0,C 180,E1 7147.709,E2 7147.709} C_VEL
LIN {X 0,Y 642.986,Z 938.368,A -85,B 0,C 180,E1 7149.895,E2 7149.895} C_VEL
LIN {X 0,Y 646.78,Z 892.163,A -85,B 0,C 180,E1 7151.596,E2 7151.596} C_VEL
LIN {X 0,Y 649.696,Z 842.577,A -85,B 0,C 180,E1 7152.801,E2 7152.801} C_VEL
LIN {X 0,Y 650.203,Z 807.856,A -85,B 0,C 180,E1 7153.385,E2 7153.385} C_VEL
LIN {X 0,Y 629.172,Z 771.827,A -85,B 0,C 180,E1 7155.676,E2 7155.676} C_VEL
LIN {X 0,Y 616.901,Z 750.408,A -85,B 0,C 180,E1 7157.068,E2 7157.068} C_VEL
LIN {X 0,Y 616.848,Z 749.56,A -85,B 0,C 180,E1 7157.3,E2 7157.3} C_VEL
LIN {X 0,Y 616.777,Z 749.56,A -85,B 0,C 180,E1 7162.233,E2 7162.233} C_VEL
LIN {X 0,Y 616.791,Z 749.56,A -85,B 0,C 180,E1 7167.388,E2 7167.388} C_VEL
LIN {X 0,Y 616.827,Z 749.56,A -85,B 0,C 180,E1 7172.263,E2 7172.263} C_VEL
LIN {X 0,Y 616.917,Z 749.56,A -85,B 0,C 180,E1 7176.93,E2 7176.93} C_VEL
LIN {X 0,Y 617.133,Z 749.56,A -85,B 0,C 180,E1 7182.737,E2 7182.737} C_VEL
LIN {X 0,Y 617.235,Z 749.56,A -85,B 0,C 180,E1 7188.315,E2 7188.315} C_VEL
LIN {X 0,Y 617.379,Z 749.56,A -85,B 0,C 180,E1 7192.974,E2 7192.974} C_VEL
LIN {X 0,Y 617.703,Z 749.56,A -85,B 0,C 180,E1 7198.602,E2 7198.602} C_VEL
LIN {X 0,Y 617.502,Z 749.56,A -85,B 0,C 180,E1 7204.214,E2 7204.214} C_VEL
LIN {X 0,Y 617.314,Z 749.56,A -85,B 0,C 180,E1 7209.871,E2 7209.871} C_VEL
LIN {X 0,Y 616.997,Z 749.56,A -85,B 0,C 180,E1 7215.633,E2 7215.633} C_VEL
LIN {X 0,Y 616.913,Z 749.56,A -85,B 0,C 180,E1 7221.562,E2 7221.562} C_VEL
LIN {X 0,Y 616.793,Z 749.56,A -85,B 0,C 180,E1 7226.172,E2 7226.172} C_VEL
LIN {X 0,Y 616.811,Z 749.56,A -85,B 0,C 180,E1 7230.968,E2 7230.968} C_VEL
LIN {X 0,Y 616.804,Z 749.56,A -85,B 0,C 180,E1 7236.054,E2 7236.054} C_VEL
LIN {X 0,Y 616.807,Z 749.56,A -85,B 0,C 180,E1 7238.864,E2 7238.864} C_VEL
LIN {X 0,Y 619.219,Z 755.24,A -85,B 0,C 180,E1 7239.192,E2 7239.192} C_VEL
LIN {X 0,Y 637.896,Z 788.52,A -85,B 0,C 180,E1 7241.388,E2 7241.388} C_VEL
LIN {X 0,Y 644.344,Z 802.636,A -85,B 0,C 180,E1 7242.238,E2 7242.238} C_VEL
LIN {X 0,Y 641.768,Z 844.767,A -85,B 0,C 180,E1 7243.347,E2 7243.347} C_VEL
LIN {X 0,Y 637.982,Z 890.746,A -85,B 0,C 180,E1 7245.138,E2 7245.138} C_VEL
LIN {X 0,Y 633.952,Z 932.51,A -85,B 0,C 180,E1 7247.327,E2 7247.327} C_VEL
LIN {X 0,Y 629.939,Z 972.788,A -85,B 0,C 180,E1 7250.078,E2 7250.078} C_VEL
LIN {X 0,Y 625.875,Z 1011.492,A -85,B 0,C 180,E1 7253.489,E2 7253.489} C_VEL
LIN {X 0,Y 622.688,Z 1043.458,A -85,B 0,C 180,E1 7257.069,E2 7257.069} C_VEL
LIN {X 0,Y 620.439,Z 1070.332,A -85,B 0,C 180,E1 7260.85,E2 7260.85} C_VEL
LIN {X 0,Y 618.87,Z 1093.186,A -85,B 0,C 180,E1 7265.029,E2 7265.029} C_VEL
LIN {X 0,Y 618.105,Z 1109.057,A -85,B 0,C 180,E1 7268.863,E2 7268.863} C_VEL
LIN {X 0,Y 617.617,Z 1120.758,A -85,B 0,C 180,E1 7272.927,E2 7272.927} C_VEL
LIN {X 0,Y 617.563,Z 1126.288,A -85,B 0,C 180,E1 7275.837,E2 7275.837} C_VEL
LIN {X 0,Y 617.479,Z 1129.81,A -85,B 0,C 180,E1 7280.137,E2 7280.137} C_VEL
LIN {X 0,Y 617.573,Z 1128.336,A -85,B 0,C 180,E1 7284.384,E2 7284.384} C_VEL
LIN {X 0,Y 617.717,Z 1123.154,A -85,B 0,C 180,E1 7287.898,E2 7287.898} C_VEL
LIN {X 0,Y 617.918,Z 1112.155,A -85,B 0,C 180,E1 7292.103,E2 7292.103} C_VEL
LIN {X 0,Y 618.7,Z 1095.927,A -85,B 0,C 180,E1 7296.311,E2 7296.311} C_VEL
LIN {X 0,Y 620.193,Z 1073.524,A -85,B 0,C 180,E1 7300.53,E2 7300.53} C_VEL
LIN {X 0,Y 622.327,Z 1046.865,A -85,B 0,C 180,E1 7304.413,E2 7304.413} C_VEL
LIN {X 0,Y 625.563,Z 1014.537,A -85,B 0,C 180,E1 7308.121,E2 7308.121} C_VEL
LIN {X 0,Y 629.535,Z 976.114,A -85,B 0,C 180,E1 7311.566,E2 7311.566} C_VEL
LIN {X 0,Y 633.552,Z 937.4,A -85,B 0,C 180,E1 7314.281,E2 7314.281} C_VEL
LIN {X 0,Y 637.744,Z 893.271,A -85,B 0,C 180,E1 7316.662,E2 7316.662} C_VEL
LIN {X 0,Y 641.649,Z 846.366,A -85,B 0,C 180,E1 7318.501,E2 7318.501} C_VEL
LIN {X 0,Y 644.156,Z 807.11,A -85,B 0,C 180,E1 7319.568,E2 7319.568} C_VEL
LIN {X 0,Y 643.61,Z 801.432,A -85,B 0,C 180,E1 7319.745,E2 7319.745} C_VEL
LIN {X 0,Y 627.413,Z 768.914,A -85,B 0,C 180,E1 7321.724,E2 7321.724} C_VEL
LIN {X 0,Y 616.942,Z 750.365,A -85,B 0,C 180,E1 7322.944,E2 7322.944} C_VEL
LIN {X 0,Y 616.775,Z 749.56,A -85,B 0,C 180,E1 7327.772,E2 7327.772} C_VEL
LIN {X 0,Y 616.894,Z 749.56,A -85,B 0,C 180,E1 7333.306,E2 7333.306} C_VEL
LIN {X 0,Y 616.812,Z 749.56,A -85,B 0,C 180,E1 7338.581,E2 7338.581} C_VEL
LIN {X 0,Y 616.789,Z 749.56,A -85,B 0,C 180,E1 7343.979,E2 7343.979} C_VEL
LIN {X 0,Y 616.789,Z 749.56,A -85,B 0,C 180,E1 7349.038,E2 7349.038} C_VEL
LIN {X 0,Y 616.804,Z 749.56,A -85,B 0,C 180,E1 7353.828,E2 7353.828} C_VEL
LIN {X 0,Y 616.889,Z 749.56,A -85,B 0,C 180,E1 7358.569,E2 7358.569} C_VEL
LIN {X 0,Y 617,Z 749.56,A -85,B 0,C 180,E1 7364.367,E2 7364.367} C_VEL
LIN {X 0,Y 617.324,Z 749.56,A -85,B 0,C 180,E1 7370.129,E2 7370.129} C_VEL
LIN {X 0,Y 617.5,Z 749.56,A -85,B 0,C 180,E1 7375.786,E2 7375.786} C_VEL
LIN {X 0,Y 617.722,Z 749.56,A -85,B 0,C 180,E1 7381.398,E2 7381.398} C_VEL
LIN {X 0,Y 617.387,Z 749.56,A -85,B 0,C 180,E1 7387.026,E2 7387.026} C_VEL
LIN {X 0,Y 617.278,Z 749.56,A -85,B 0,C 180,E1 7392.724,E2 7392.724} C_VEL
LIN {X 0,Y 617.217,Z 749.56,A -85,B 0,C 180,E1 7397.284,E2 7397.284} C_VEL
LIN {X 0,Y 617.134,Z 749.56,A -85,B 0,C 180,E1 7401.545,E2 7401.545} C_VEL
LIN {X 0,Y 617.058,Z 749.56,A -85,B 0,C 180,E1 7406.152,E2 7406.152} C_VEL
LIN {X 0,Y 616.923,Z 749.56,A -85,B 0,C 180,E1 7410.983,E2 7410.983} C_VEL
LIN {X 0,Y 616.843,Z 749.56,A -85,B 0,C 180,E1 7416.056,E2 7416.056} C_VEL
LIN {X 0,Y 616.845,Z 749.56,A -85,B 0,C 180,E1 7421.406,E2 7421.406} C_VEL
LIN {X 0,Y 616.92,Z 749.965,A -85,B 0,C 180,E1 7422.895,E2 7422.895} C_VEL
LIN {X 0,Y 619.625,Z 755.525,A -85,B 0,C 180,E1 7423.227,E2 7423.227} C_VEL
LIN {X 0,Y 632.48,Z 777.088,A -85,B 0,C 180,E1 7424.666,E2 7424.666} C_VEL
LIN {X 0,Y 635.592,Z 784.244,A -85,B 0,C 180,E1 7425.029,E2 7425.029} C_VEL
LIN {X 0,Y 641.734,Z 805.825,A -85,B 0,C 180,E1 7425.865,E2 7425.865} C_VEL
LIN {X 0,Y 642.642,Z 807.452,A -85,B 0,C 180,E1 7425.969,E2 7425.969} C_VEL
LIN {X 0,Y 644.939,Z 812.304,A -85,B 0,C 180,E1 7426.239,E2 7426.239} C_VEL
LIN {X 0,Y 642.877,Z 863.067,A -85,B 0,C 180,E1 7427.157,E2 7427.157} C_VEL
LIN {X 0,Y 639.424,Z 908.189,A -85,B 0,C 180,E1 7428.452,E2 7428.452} C_VEL
LIN {X 0,Y 635.248,Z 954.109,A -85,B 0,C 180,E1 7430.354,E2 7430.354} C_VEL
LIN {X 0,Y 630.151,Z 999.535,A -85,B 0,C 180,E1 7432.879,E2 7432.879} C_VEL
LIN {X 0,Y 625.266,Z 1040.256,A -85,B 0,C 180,E1 7435.79,E2 7435.79} C_VEL
LIN {X 0,Y 620.295,Z 1080.24,A -85,B 0,C 180,E1 7439.413,E2 7439.413} C_VEL
LIN {X 0,Y 616.401,Z 1113.629,A -85,B 0,C 180,E1 7443.209,E2 7443.209} C_VEL
LIN {X 0,Y 613.347,Z 1144.517,A -85,B 0,C 180,E1 7447.625,E2 7447.625} C_VEL
LIN {X 0,Y 611.469,Z 1168.58,A -85,B 0,C 180,E1 7452.079,E2 7452.079} C_VEL
LIN {X 0,Y 610.409,Z 1186.375,A -85,B 0,C 180,E1 7456.397,E2 7456.397} C_VEL
LIN {X 0,Y 609.889,Z 1199.102,A -85,B 0,C 180,E1 7460.731,E2 7460.731} C_VEL
LIN {X 0,Y 609.758,Z 1205.909,A -85,B 0,C 180,E1 7464.31,E2 7464.31} C_VEL
LIN {X 0,Y 609.647,Z 1209.667,A -85,B 0,C 180,E1 7468.579,E2 7468.579} C_VEL
LIN {X 0,Y 609.8,Z 1208.928,A -85,B 0,C 180,E1 7472.84,E2 7472.84} C_VEL
LIN {X 0,Y 609.801,Z 1203.568,A -85,B 0,C 180,E1 7477.117,E2 7477.117} C_VEL
LIN {X 0,Y 610.062,Z 1193.421,A -85,B 0,C 180,E1 7481.429,E2 7481.429} C_VEL
LIN {X 0,Y 610.745,Z 1178.009,A -85,B 0,C 180,E1 7485.792,E2 7485.792} C_VEL
LIN {X 0,Y 612.034,Z 1158.941,A -85,B 0,C 180,E1 7489.845,E2 7489.845} C_VEL
LIN {X 0,Y 614.248,Z 1133.815,A -85,B 0,C 180,E1 7494.038,E2 7494.038} C_VEL
LIN {X 0,Y 617.661,Z 1102.385,A -85,B 0,C 180,E1 7498.162,E2 7498.162} C_VEL
LIN {X 0,Y 621.961,Z 1066.642,A -85,B 0,C 180,E1 7501.919,E2 7501.919} C_VEL
LIN {X 0,Y 626.989,Z 1025.611,A -85,B 0,C 180,E1 7505.34,E2 7505.34} C_VEL
LIN {X 0,Y 631.938,Z 984.663,A -85,B 0,C 180,E1 7508.024,E2 7508.024} C_VEL
LIN {X 0,Y 636.703,Z 939.33,A -85,B 0,C 180,E1 7510.318,E2 7510.318} C_VEL
LIN {X 0,Y 640.714,Z 893.632,A -85,B 0,C 180,E1 7512.027,E2 7512.027} C_VEL
LIN {X 0,Y 643.817,Z 843.812,A -85,B 0,C 180,E1 7513.258,E2 7513.258} C_VEL
LIN {X 0,Y 644.541,Z 811.191,A -85,B 0,C 180,E1 7513.812,E2 7513.812} C_VEL
LIN {X 0,Y 617.406,Z 765.473,A -85,B 0,C 180,E1 7516.785,E2 7516.785} C_VEL
LIN {X 0,Y 608.985,Z 750.673,A -85,B 0,C 180,E1 7517.781,E2 7517.781} C_VEL
LIN {X 0,Y 608.914,Z 749.56,A -85,B 0,C 180,E1 7517.933,E2 7517.933} C_VEL
LIN {X 0,Y 608.863,Z 749.56,A -85,B 0,C 180,E1 7523.445,E2 7523.445} C_VEL
LIN {X 0,Y 608.885,Z 749.56,A -85,B 0,C 180,E1 7528.593,E2 7528.593} C_VEL
LIN {X 0,Y 608.94,Z 749.56,A -85,B 0,C 180,E1 7533.473,E2 7533.473} C_VEL
LIN {X 0,Y 609.021,Z 749.56,A -85,B 0,C 180,E1 7538.153,E2 7538.153} C_VEL
LIN {X 0,Y 609.235,Z 749.56,A -85,B 0,C 180,E1 7542.688,E2 7542.688} C_VEL
LIN {X 0,Y 609.347,Z 749.56,A -85,B 0,C 180,E1 7547.107,E2 7547.107} C_VEL
LIN {X 0,Y 609.469,Z 749.56,A -85,B 0,C 180,E1 7552.882,E2 7552.882} C_VEL
LIN {X 0,Y 609.796,Z 749.56,A -85,B 0,C 180,E1 7558.584,E2 7558.584} C_VEL
LIN {X 0,Y 609.591,Z 749.56,A -85,B 0,C 180,E1 7564.269,E2 7564.269} C_VEL
LIN {X 0,Y 609.521,Z 749.56,A -85,B 0,C 180,E1 7568.559,E2 7568.559} C_VEL
LIN {X 0,Y 609.134,Z 749.56,A -85,B 0,C 180,E1 7574.368,E2 7574.368} C_VEL
LIN {X 0,Y 609.003,Z 749.56,A -85,B 0,C 180,E1 7580.332,E2 7580.332} C_VEL
LIN {X 0,Y 608.894,Z 749.56,A -85,B 0,C 180,E1 7584.96,E2 7584.96} C_VEL
LIN {X 0,Y 608.895,Z 749.56,A -85,B 0,C 180,E1 7589.764,E2 7589.764} C_VEL
LIN {X 0,Y 608.845,Z 749.56,A -85,B 0,C 180,E1 7595.012,E2 7595.012} C_VEL
LIN {X 0,Y 608.89,Z 749.956,A -85,B 0,C 180,E1 7598.105,E2 7598.105} C_VEL
LIN {X 0,Y 611.528,Z 755.463,A -85,B 0,C 180,E1 7598.46,E2 7598.46} C_VEL
LIN {X 0,Y 631.654,Z 790.95,A -85,B 0,C 180,E1 7600.918,E2 7600.918} C_VEL
LIN {X 0,Y 638.365,Z 806.426,A -85,B 0,C 180,E1 7601.844,E2 7601.844} C_VEL
LIN {X 0,Y 635.527,Z 847.626,A -85,B 0,C 180,E1 7602.967,E2 7602.967} C_VEL
LIN {X 0,Y 631.814,Z 889.578,A -85,B 0,C 180,E1 7604.628,E2 7604.628} C_VEL
LIN {X 0,Y 627.025,Z 934.177,A -85,B 0,C 180,E1 7607.018,E2 7607.018} C_VEL
LIN {X 0,Y 622.796,Z 973.811,A -85,B 0,C 180,E1 7609.775,E2 7609.775} C_VEL
LIN {X 0,Y 618.537,Z 1011.885,A -85,B 0,C 180,E1 7613.176,E2 7613.176} C_VEL
LIN {X 0,Y 615.224,Z 1043.125,A -85,B 0,C 180,E1 7616.716,E2 7616.716} C_VEL
LIN {X 0,Y 612.679,Z 1071.193,A -85,B 0,C 180,E1 7620.73,E2 7620.73} C_VEL
LIN {X 0,Y 611.057,Z 1093.629,A -85,B 0,C 180,E1 7624.914,E2 7624.914} C_VEL
LIN {X 0,Y 610.236,Z 1109.909,A -85,B 0,C 180,E1 7628.958,E2 7628.958} C_VEL
LIN {X 0,Y 609.764,Z 1120.491,A -85,B 0,C 180,E1 7632.7,E2 7632.7} C_VEL
LIN {X 0,Y 609.661,Z 1126.104,A -85,B 0,C 180,E1 7635.65,E2 7635.65} C_VEL
LIN {X 0,Y 609.556,Z 1129.781,A -85,B 0,C 180,E1 7640.007,E2 7640.007} C_VEL
LIN {X 0,Y 609.665,Z 1128.426,A -85,B 0,C 180,E1 7644.311,E2 7644.311} C_VEL
LIN {X 0,Y 609.827,Z 1123.38,A -85,B 0,C 180,E1 7647.871,E2 7647.871} C_VEL
LIN {X 0,Y 610.06,Z 1112.53,A -85,B 0,C 180,E1 7652.13,E2 7652.13} C_VEL
LIN {X 0,Y 610.871,Z 1096.457,A -85,B 0,C 180,E1 7656.392,E2 7656.392} C_VEL
LIN {X 0,Y 612.448,Z 1074.234,A -85,B 0,C 180,E1 7660.665,E2 7660.665} C_VEL
LIN {X 0,Y 614.716,Z 1047.816,A -85,B 0,C 180,E1 7664.595,E2 7664.595} C_VEL
LIN {X 0,Y 618.375,Z 1013.984,A -85,B 0,C 180,E1 7668.524,E2 7668.524} C_VEL
LIN {X 0,Y 622.582,Z 975.419,A -85,B 0,C 180,E1 7672.006,E2 7672.006} C_VEL
LIN {X 0,Y 626.871,Z 936.099,A -85,B 0,C 180,E1 7674.771,E2 7674.771} C_VEL
LIN {X 0,Y 631.674,Z 889.792,A -85,B 0,C 180,E1 7677.273,E2 7677.273} C_VEL
LIN {X 0,Y 635.798,Z 843.832,A -85,B 0,C 180,E1 7679.059,E2 7679.059} C_VEL
LIN {X 0,Y 637.786,Z 804.936,A -85,B 0,C 180,E1 7680.128,E2 7680.128} C_VEL
LIN {X 0,Y 621.744,Z 772.306,A -85,B 0,C 180,E1 7682.165,E2 7682.165} C_VEL
LIN {X 0,Y 609.138,Z 751.212,A -85,B 0,C 180,E1 7683.646,E2 7683.646} C_VEL
LIN {X 0,Y 608.949,Z 749.56,A -85,B 0,C 180,E1 7683.722,E2 7683.722} C_VEL
LIN {X 0,Y 608.887,Z 749.56,A -85,B 0,C 180,E1 7689.696,E2 7689.696} C_VEL
LIN {X 0,Y 608.941,Z 749.56,A -85,B 0,C 180,E1 7694.015,E2 7694.015} C_VEL
LIN {X 0,Y 608.874,Z 749.56,A -85,B 0,C 180,E1 7699.807,E2 7699.807} C_VEL
LIN {X 0,Y 608.816,Z 749.56,A -85,B 0,C 180,E1 7705.183,E2 7705.183} C_VEL
LIN {X 0,Y 608.858,Z 749.56,A -85,B 0,C 180,E1 7710.305,E2 7710.305} C_VEL
LIN {X 0,Y 608.898,Z 749.56,A -85,B 0,C 180,E1 7715.041,E2 7715.041} C_VEL
LIN {X 0,Y 608.966,Z 749.56,A -85,B 0,C 180,E1 7720.556,E2 7720.556} C_VEL
LIN {X 0,Y 609.133,Z 749.56,A -85,B 0,C 180,E1 7725.632,E2 7725.632} C_VEL
LIN {X 0,Y 609.405,Z 749.56,A -85,B 0,C 180,E1 7730,E2 7730} C_VEL
LIN {X 0,Y 609.589,Z 749.56,A -85,B 0,C 180,E1 7735.731,E2 7735.731} C_VEL
LIN {X 0,Y 609.814,Z 749.56,A -85,B 0,C 180,E1 7741.416,E2 7741.416} C_VEL
LIN {X 0,Y 609.475,Z 749.56,A -85,B 0,C 180,E1 7747.357,E2 7747.357} C_VEL
LIN {X 0,Y 609.354,Z 749.56,A -85,B 0,C 180,E1 7752.893,E2 7752.893} C_VEL
LIN {X 0,Y 609.321,Z 749.56,A -85,B 0,C 180,E1 7757.31,E2 7757.31} C_VEL
LIN {X 0,Y 609.188,Z 749.56,A -85,B 0,C 180,E1 7761.841,E2 7761.841} C_VEL
LIN {X 0,Y 609.084,Z 749.56,A -85,B 0,C 180,E1 7766.726,E2 7766.726} C_VEL
LIN {X 0,Y 609.006,Z 749.56,A -85,B 0,C 180,E1 7772.472,E2 7772.472} C_VEL
LIN {X 0,Y 608.899,Z 749.56,A -85,B 0,C 180,E1 7778.344,E2 7778.344} C_VEL
LIN {X 0,Y 608.952,Z 749.56,A -85,B 0,C 180,E1 7782.143,E2 7782.143} C_VEL
LIN {X 0,Y 611.49,Z 755.287,A -85,B 0,C 180,E1 7782.484,E2 7782.484} C_VEL
LIN {X 0,Y 642.642,Z 807.452,A -85,B 0,C 180,E1 7785.969,E2 7785.969} C_VEL
LIN {X 0,Y 643.206,Z 814.029,A -85,B 0,C 180,E1 7786.117,E2 7786.117} C_VEL
LIN {X 0,Y 638.733,Z 830.817,A -85,B 0,C 180,E1 7786.03,E2 7786.03} C_VEL
LIN {X 0,Y 635.808,Z 879.361,A -85,B 0,C 180,E1 7787.069,E2 7787.069} C_VEL
LIN {X 0,Y 631.836,Z 926.216,A -85,B 0,C 180,E1 7788.654,E2 7788.654} C_VEL
LIN {X 0,Y 626.993,Z 971.919,A -85,B 0,C 180,E1 7790.792,E2 7790.792} C_VEL
LIN {X 0,Y 621.289,Z 1017.517,A -85,B 0,C 180,E1 7793.631,E2 7793.631} C_VEL
LIN {X 0,Y 616.139,Z 1057.668,A -85,B 0,C 180,E1 7796.849,E2 7796.849} C_VEL
LIN {X 0,Y 611.222,Z 1096.197,A -85,B 0,C 180,E1 7800.744,E2 7800.744} C_VEL
LIN {X 0,Y 607.327,Z 1129.138,A -85,B 0,C 180,E1 7804.976,E2 7804.976} C_VEL
LIN {X 0,Y 604.772,Z 1154.987,A -85,B 0,C 180,E1 7809.141,E2 7809.141} C_VEL
LIN {X 0,Y 603.028,Z 1176.472,A -85,B 0,C 180,E1 7813.625,E2 7813.625} C_VEL
LIN {X 0,Y 602.21,Z 1192.518,A -85,B 0,C 180,E1 7818.121,E2 7818.121} C_VEL
LIN {X 0,Y 601.888,Z 1202.693,A -85,B 0,C 180,E1 7822.298,E2 7822.298} C_VEL
LIN {X 0,Y 601.793,Z 1207.677,A -85,B 0,C 180,E1 7825.679,E2 7825.679} C_VEL
LIN {X 0,Y 601.859,Z 1210,A -85,B 0,C 180,E1 7829.999,E2 7829.999} C_VEL
LIN {X 0,Y 601.785,Z 1207.679,A -85,B 0,C 180,E1 7834.32,E2 7834.32} C_VEL
LIN {X 0,Y 601.89,Z 1200.693,A -85,B 0,C 180,E1 7838.663,E2 7838.663} C_VEL
LIN {X 0,Y 602.344,Z 1188.888,A -85,B 0,C 180,E1 7843.048,E2 7843.048} C_VEL
LIN {X 0,Y 603.445,Z 1171.707,A -85,B 0,C 180,E1 7847.487,E2 7847.487} C_VEL
LIN {X 0,Y 605.335,Z 1148.501,A -85,B 0,C 180,E1 7851.99,E2 7851.99} C_VEL
LIN {X 0,Y 608.284,Z 1121.045,A -85,B 0,C 180,E1 7856.164,E2 7856.164} C_VEL
LIN {X 0,Y 612.446,Z 1086.025,A -85,B 0,C 180,E1 7860.375,E2 7860.375} C_VEL
LIN {X 0,Y 617.237,Z 1048.776,A -85,B 0,C 180,E1 7863.931,E2 7863.931} C_VEL
LIN {X 0,Y 622.715,Z 1006.726,A -85,B 0,C 180,E1 7867.116,E2 7867.116} C_VEL
LIN {X 0,Y 627.999,Z 962.651,A -85,B 0,C 180,E1 7869.69,E2 7869.69} C_VEL
LIN {X 0,Y 632.927,Z 915.144,A -85,B 0,C 180,E1 7871.78,E2 7871.78} C_VEL
LIN {X 0,Y 636.632,Z 868.401,A -85,B 0,C 180,E1 7873.208,E2 7873.208} C_VEL
LIN {X 0,Y 639.083,Z 820.325,A -85,B 0,C 180,E1 7874.13,E2 7874.13} C_VEL
LIN {X 0,Y 638.37,Z 813.646,A -85,B 0,C 180,E1 7874.307,E2 7874.307} C_VEL
LIN {X 0,Y 603.292,Z 755.099,A -85,B 0,C 180,E1 7878.248,E2 7878.248} C_VEL
LIN {X 0,Y 600.944,Z 749.56,A -85,B 0,C 180,E1 7878.629,E2 7878.629} C_VEL
LIN {X 0,Y 600.944,Z 749.56,A -85,B 0,C 180,E1 7883.577,E2 7883.577} C_VEL
LIN {X 0,Y 600.966,Z 749.56,A -85,B 0,C 180,E1 7888.75,E2 7888.75} C_VEL
LIN {X 0,Y 601.011,Z 749.56,A -85,B 0,C 180,E1 7893.095,E2 7893.095} C_VEL
LIN {X 0,Y 601.109,Z 749.56,A -85,B 0,C 180,E1 7898.455,E2 7898.455} C_VEL
LIN {X 0,Y 601.345,Z 749.56,A -85,B 0,C 180,E1 7903.957,E2 7903.957} C_VEL
LIN {X 0,Y 601.462,Z 749.56,A -85,B 0,C 180,E1 7908.474,E2 7908.474} C_VEL
LIN {X 0,Y 601.669,Z 749.56,A -85,B 0,C 180,E1 7914.238,E2 7914.238} C_VEL
LIN {X 0,Y 601.855,Z 749.56,A -85,B 0,C 180,E1 7920.004,E2 7920.004} C_VEL
LIN {X 0,Y 601.694,Z 749.56,A -85,B 0,C 180,E1 7924.325,E2 7924.325} C_VEL
LIN {X 0,Y 601.596,Z 749.56,A -85,B 0,C 180,E1 7928.672,E2 7928.672} C_VEL
LIN {X 0,Y 601.305,Z 749.56,A -85,B 0,C 180,E1 7933.077,E2 7933.077} C_VEL
LIN {X 0,Y 601.06,Z 749.56,A -85,B 0,C 180,E1 7939.081,E2 7939.081} C_VEL
LIN {X 0,Y 600.964,Z 749.56,A -85,B 0,C 180,E1 7943.728,E2 7943.728} C_VEL
LIN {X 0,Y 600.976,Z 749.56,A -85,B 0,C 180,E1 7948.544,E2 7948.544} C_VEL
LIN {X 0,Y 600.895,Z 749.56,A -85,B 0,C 180,E1 7953.915,E2 7953.915} C_VEL
LIN {X 0,Y 600.976,Z 749.898,A -85,B 0,C 180,E1 7957.288,E2 7957.288} C_VEL
LIN {X 0,Y 603.504,Z 755.353,A -85,B 0,C 180,E1 7957.648,E2 7957.648} C_VEL
LIN {X 0,Y 624.669,Z 791.707,A -85,B 0,C 180,E1 7960.33,E2 7960.33} C_VEL
LIN {X 0,Y 632.319,Z 808.787,A -85,B 0,C 180,E1 7961.408,E2 7961.408} C_VEL
LIN {X 0,Y 629.16,Z 851.929,A -85,B 0,C 180,E1 7962.627,E2 7962.627} C_VEL
LIN {X 0,Y 625.278,Z 893.644,A -85,B 0,C 180,E1 7964.335,E2 7964.335} C_VEL
LIN {X 0,Y 620.297,Z 935.23,A -85,B 0,C 180,E1 7966.647,E2 7966.647} C_VEL
LIN {X 0,Y 615.508,Z 976.086,A -85,B 0,C 180,E1 7969.567,E2 7969.567} C_VEL
LIN {X 0,Y 611.091,Z 1013.642,A -85,B 0,C 180,E1 7972.992,E2 7972.992} C_VEL
LIN {X 0,Y 607.283,Z 1047.486,A -85,B 0,C 180,E1 7976.964,E2 7976.964} C_VEL
LIN {X 0,Y 604.73,Z 1074.373,A -85,B 0,C 180,E1 7981.008,E2 7981.008} C_VEL
LIN {X 0,Y 603.11,Z 1095.903,A -85,B 0,C 180,E1 7985.186,E2 7985.186} C_VEL
LIN {X 0,Y 602.282,Z 1111.911,A -85,B 0,C 180,E1 7989.436,E2 7989.436} C_VEL
LIN {X 0,Y 601.833,Z 1121.962,A -85,B 0,C 180,E1 7993.275,E2 7993.275} C_VEL
LIN {X 0,Y 601.647,Z 1127.756,A -85,B 0,C 180,E1 7996.936,E2 7996.936} C_VEL
LIN {X 0,Y 601.741,Z 1129.918,A -85,B 0,C 180,E1 8001.335,E2 8001.335} C_VEL
LIN {X 0,Y 601.835,Z 1126.914,A -85,B 0,C 180,E1 8005.681,E2 8005.681} C_VEL
LIN {X 0,Y 602.091,Z 1118.91,A -85,B 0,C 180,E1 8010.001,E2 8010.001} C_VEL
LIN {X 0,Y 602.62,Z 1105.603,A -85,B 0,C 180,E1 8014.315,E2 8014.315} C_VEL
LIN {X 0,Y 603.757,Z 1086.756,A -85,B 0,C 180,E1 8018.638,E2 8018.638} C_VEL
LIN {X 0,Y 605.828,Z 1061.509,A -85,B 0,C 180,E1 8022.974,E2 8022.974} C_VEL
LIN {X 0,Y 608.954,Z 1032.094,A -85,B 0,C 180,E1 8026.868,E2 8026.868} C_VEL
LIN {X 0,Y 612.817,Z 999.205,A -85,B 0,C 180,E1 8030.333,E2 8030.333} C_VEL
LIN {X 0,Y 617.485,Z 960.015,A -85,B 0,C 180,E1 8033.574,E2 8033.574} C_VEL
LIN {X 0,Y 622.661,Z 916.258,A -85,B 0,C 180,E1 8036.387,E2 8036.387} C_VEL
LIN {X 0,Y 627.023,Z 874.462,A -85,B 0,C 180,E1 8038.421,E2 8038.421} C_VEL
LIN {X 0,Y 630.982,Z 825.643,A -85,B 0,C 180,E1 8040.087,E2 8040.087} C_VEL
LIN {X 0,Y 631.743,Z 807.902,A -85,B 0,C 180,E1 8040.548,E2 8040.548} C_VEL
LIN {X 0,Y 616.955,Z 777.472,A -85,B 0,C 180,E1 8042.496,E2 8042.496} C_VEL
LIN {X 0,Y 601.219,Z 751.418,A -85,B 0,C 180,E1 8044.385,E2 8044.385} C_VEL
LIN {X 0,Y 601.001,Z 749.56,A -85,B 0,C 180,E1 8044.491,E2 8044.491} C_VEL
LIN {X 0,Y 600.942,Z 749.56,A -85,B 0,C 180,E1 8048.951,E2 8048.951} C_VEL
LIN {X 0,Y 600.95,Z 749.56,A -85,B 0,C 180,E1 8054.756,E2 8054.756} C_VEL
LIN {X 0,Y 600.917,Z 749.56,A -85,B 0,C 180,E1 8059.163,E2 8059.163} C_VEL
LIN {X 0,Y 600.916,Z 749.56,A -85,B 0,C 180,E1 8064.657,E2 8064.657} C_VEL
LIN {X 0,Y 600.893,Z 749.56,A -85,B 0,C 180,E1 8069.799,E2 8069.799} C_VEL
LIN {X 0,Y 600.969,Z 749.56,A -85,B 0,C 180,E1 8074.854,E2 8074.854} C_VEL
LIN {X 0,Y 601.043,Z 749.56,A -85,B 0,C 180,E1 8079.386,E2 8079.386} C_VEL
LIN {X 0,Y 601.217,Z 749.56,A -85,B 0,C 180,E1 8085.438,E2 8085.438} C_VEL
LIN {X 0,Y 601.483,Z 749.56,A -85,B 0,C 180,E1 8089.867,E2 8089.867} C_VEL
LIN {X 0,Y 601.605,Z 749.56,A -85,B 0,C 180,E1 8094.229,E2 8094.229} C_VEL
LIN {X 0,Y 601.736,Z 749.56,A -85,B 0,C 180,E1 8098.557,E2 8098.557} C_VEL
LIN {X 0,Y 601.67,Z 749.56,A -85,B 0,C 180,E1 8102.875,E2 8102.875} C_VEL
LIN {X 0,Y 601.594,Z 749.56,A -85,B 0,C 180,E1 8107.211,E2 8107.211} C_VEL
LIN {X 0,Y 601.452,Z 749.56,A -85,B 0,C 180,E1 8113.065,E2 8113.065} C_VEL
LIN {X 0,Y 601.395,Z 749.56,A -85,B 0,C 180,E1 8117.545,E2 8117.545} C_VEL
LIN {X 0,Y 601.246,Z 749.56,A -85,B 0,C 180,E1 8122.144,E2 8122.144} C_VEL
LIN {X 0,Y 601.185,Z 749.56,A -85,B 0,C 180,E1 8126.897,E2 8126.897} C_VEL
LIN {X 0,Y 601.078,Z 749.56,A -85,B 0,C 180,E1 8131.863,E2 8131.863} C_VEL
LIN {X 0,Y 600.969,Z 749.56,A -85,B 0,C 180,E1 8137.115,E2 8137.115} C_VEL
LIN {X 0,Y 600.975,Z 749.56,A -85,B 0,C 180,E1 8141.372,E2 8141.372} C_VEL
LIN {X 0,Y 603.548,Z 755.348,A -85,B 0,C 180,E1 8141.733,E2 8141.733} C_VEL
LIN {X 0,Y 639.183,Z 814.877,A -85,B 0,C 180,E1 8145.782,E2 8145.782} C_VEL
LIN {X 0,Y 638.733,Z 830.817,A -85,B 0,C 180,E1 8146.03,E2 8146.03} C_VEL
LIN {X 0,Y 635.158,Z 847.976,A -85,B 0,C 180,E1 8146.1,E2 8146.1} C_VEL
LIN {X 0,Y 631.37,Z 862.855,A -85,B 0,C 180,E1 8146.179,E2 8146.179} C_VEL
LIN {X 0,Y 631.146,Z 864.986,A -85,B 0,C 180,E1 8146.224,E2 8146.224} C_VEL
LIN {X 0,Y 627.28,Z 911.055,A -85,B 0,C 180,E1 8147.582,E2 8147.582} C_VEL
LIN {X 0,Y 622.597,Z 956.189,A -85,B 0,C 180,E1 8149.509,E2 8149.509} C_VEL
LIN {X 0,Y 616.825,Z 1002.425,A -85,B 0,C 180,E1 8152.147,E2 8152.147} C_VEL
LIN {X 0,Y 611.528,Z 1041.496,A -85,B 0,C 180,E1 8155.027,E2 8155.027} C_VEL
LIN {X 0,Y 605.893,Z 1081.832,A -85,B 0,C 180,E1 8158.778,E2 8158.778} C_VEL
LIN {X 0,Y 601.46,Z 1115.209,A -85,B 0,C 180,E1 8162.708,E2 8162.708} C_VEL
LIN {X 0,Y 598.13,Z 1144.778,A -85,B 0,C 180,E1 8167.068,E2 8167.068} C_VEL
LIN {X 0,Y 595.975,Z 1168.283,A -85,B 0,C 180,E1 8171.532,E2 8171.532} C_VEL
LIN {X 0,Y 594.771,Z 1186.374,A -85,B 0,C 180,E1 8176.032,E2 8176.032} C_VEL
LIN {X 0,Y 594.143,Z 1199.102,A -85,B 0,C 180,E1 8180.483,E2 8180.483} C_VEL
LIN {X 0,Y 593.972,Z 1205.909,A -85,B 0,C 180,E1 8184.158,E2 8184.158} C_VEL
LIN {X 0,Y 593.849,Z 1209.667,A -85,B 0,C 180,E1 8188.541,E2 8188.541} C_VEL
LIN {X 0,Y 593.997,Z 1208.922,A -85,B 0,C 180,E1 8192.916,E2 8192.916} C_VEL
LIN {X 0,Y 594.011,Z 1203.563,A -85,B 0,C 180,E1 8197.307,E2 8197.307} C_VEL
LIN {X 0,Y 594.323,Z 1193.421,A -85,B 0,C 180,E1 8201.736,E2 8201.736} C_VEL
LIN {X 0,Y 595.13,Z 1178.007,A -85,B 0,C 180,E1 8206.218,E2 8206.218} C_VEL
LIN {X 0,Y 596.863,Z 1156.97,A -85,B 0,C 180,E1 8210.759,E2 8210.759} C_VEL
LIN {X 0,Y 599.501,Z 1131.677,A -85,B 0,C 180,E1 8214.991,E2 8214.991} C_VEL
LIN {X 0,Y 603.531,Z 1099.292,A -85,B 0,C 180,E1 8219.278,E2 8219.278} C_VEL
LIN {X 0,Y 608.324,Z 1064.083,A -85,B 0,C 180,E1 8222.981,E2 8222.981} C_VEL
LIN {X 0,Y 613.977,Z 1023.244,A -85,B 0,C 180,E1 8226.41,E2 8226.41} C_VEL
LIN {X 0,Y 619.572,Z 981.346,A -85,B 0,C 180,E1 8229.142,E2 8229.142} C_VEL
LIN {X 0,Y 624.743,Z 937.353,A -85,B 0,C 180,E1 8231.362,E2 8231.362} C_VEL
LIN {X 0,Y 628.962,Z 893.472,A -85,B 0,C 180,E1 8233.004,E2 8233.004} C_VEL
LIN {X 0,Y 632.075,Z 846.586,A -85,B 0,C 180,E1 8234.178,E2 8234.178} C_VEL
LIN {X 0,Y 632.789,Z 817.445,A -85,B 0,C 180,E1 8234.693,E2 8234.693} C_VEL
LIN {X 0,Y 595.483,Z 755.289,A -85,B 0,C 180,E1 8239.029,E2 8239.029} C_VEL
LIN {X 0,Y 592.993,Z 749.56,A -85,B 0,C 180,E1 8239.392,E2 8239.392} C_VEL
LIN {X 0,Y 593.034,Z 749.56,A -85,B 0,C 180,E1 8244.626,E2 8244.626} C_VEL
LIN {X 0,Y 593.041,Z 749.56,A -85,B 0,C 180,E1 8250.036,E2 8250.036} C_VEL
LIN {X 0,Y 593.098,Z 749.56,A -85,B 0,C 180,E1 8254.337,E2 8254.337} C_VEL
LIN {X 0,Y 593.229,Z 749.56,A -85,B 0,C 180,E1 8259.111,E2 8259.111} C_VEL
LIN {X 0,Y 593.432,Z 749.56,A -85,B 0,C 180,E1 8263.737,E2 8263.737} C_VEL
LIN {X 0,Y 593.523,Z 749.56,A -85,B 0,C 180,E1 8268.251,E2 8268.251} C_VEL
LIN {X 0,Y 593.696,Z 749.56,A -85,B 0,C 180,E1 8273.049,E2 8273.049} C_VEL
LIN {X 0,Y 593.982,Z 749.56,A -85,B 0,C 180,E1 8278.546,E2 8278.546} C_VEL
LIN {X 0,Y 593.782,Z 749.56,A -85,B 0,C 180,E1 8284.383,E2 8284.383} C_VEL
LIN {X 0,Y 593.696,Z 749.56,A -85,B 0,C 180,E1 8288.789,E2 8288.789} C_VEL
LIN {X 0,Y 593.339,Z 749.56,A -85,B 0,C 180,E1 8294.584,E2 8294.584} C_VEL
LIN {X 0,Y 593.173,Z 749.56,A -85,B 0,C 180,E1 8300.9,E2 8300.9} C_VEL
LIN {X 0,Y 593.049,Z 749.56,A -85,B 0,C 180,E1 8306.898,E2 8306.898} C_VEL
LIN {X 0,Y 592.969,Z 749.56,A -85,B 0,C 180,E1 8312.758,E2 8312.758} C_VEL
LIN {X 0,Y 593.066,Z 750.057,A -85,B 0,C 180,E1 8316.432,E2 8316.432} C_VEL
LIN {X 0,Y 595.801,Z 755.564,A -85,B 0,C 180,E1 8316.832,E2 8316.832} C_VEL
LIN {X 0,Y 618.416,Z 793.918,A -85,B 0,C 180,E1 8319.824,E2 8319.824} C_VEL
LIN {X 0,Y 626.229,Z 813.214,A -85,B 0,C 180,E1 8321.021,E2 8321.021} C_VEL
LIN {X 0,Y 623.033,Z 854.552,A -85,B 0,C 180,E1 8322.229,E2 8322.229} C_VEL
LIN {X 0,Y 618.839,Z 896.432,A -85,B 0,C 180,E1 8323.981,E2 8323.981} C_VEL
LIN {X 0,Y 613.388,Z 939.981,A -85,B 0,C 180,E1 8326.474,E2 8326.474} C_VEL
LIN {X 0,Y 607.65,Z 982.734,A -85,B 0,C 180,E1 8329.717,E2 8329.717} C_VEL
LIN {X 0,Y 603.357,Z 1017.556,A -85,B 0,C 180,E1 8333.053,E2 8333.053} C_VEL
LIN {X 0,Y 599.589,Z 1049.446,A -85,B 0,C 180,E1 8336.902,E2 8336.902} C_VEL
LIN {X 0,Y 596.981,Z 1075.423,A -85,B 0,C 180,E1 8340.925,E2 8340.925} C_VEL
LIN {X 0,Y 595.23,Z 1097.005,A -85,B 0,C 180,E1 8345.236,E2 8345.236} C_VEL
LIN {X 0,Y 594.38,Z 1113.25,A -85,B 0,C 180,E1 8349.715,E2 8349.715} C_VEL
LIN {X 0,Y 593.919,Z 1123.184,A -85,B 0,C 180,E1 8353.748,E2 8353.748} C_VEL
LIN {X 0,Y 593.708,Z 1128.95,A -85,B 0,C 180,E1 8358.252,E2 8358.252} C_VEL
LIN {X 0,Y 593.875,Z 1129.601,A -85,B 0,C 180,E1 8362.691,E2 8362.691} C_VEL
LIN {X 0,Y 594.059,Z 1124.981,A -85,B 0,C 180,E1 8367.085,E2 8367.085} C_VEL
LIN {X 0,Y 594.241,Z 1115.431,A -85,B 0,C 180,E1 8371.458,E2 8371.458} C_VEL
LIN {X 0,Y 594.958,Z 1101.952,A -85,B 0,C 180,E1 8375.466,E2 8375.466} C_VEL
LIN {X 0,Y 596.339,Z 1081.748,A -85,B 0,C 180,E1 8379.849,E2 8379.849} C_VEL
LIN {X 0,Y 598.67,Z 1057.1,A -85,B 0,C 180,E1 8383.916,E2 8383.916} C_VEL
LIN {X 0,Y 602.368,Z 1026.28,A -85,B 0,C 180,E1 8387.898,E2 8387.898} C_VEL
LIN {X 0,Y 607.037,Z 988.086,A -85,B 0,C 180,E1 8391.734,E2 8391.734} C_VEL
LIN {X 0,Y 612.95,Z 943.372,A -85,B 0,C 180,E1 8395.203,E2 8395.203} C_VEL
LIN {X 0,Y 617.909,Z 902.834,A -85,B 0,C 180,E1 8397.59,E2 8397.59} C_VEL
LIN {X 0,Y 622.305,Z 862.14,A -85,B 0,C 180,E1 8399.386,E2 8399.386} C_VEL
LIN {X 0,Y 625.662,Z 817.919,A -85,B 0,C 180,E1 8400.76,E2 8400.76} C_VEL
LIN {X 0,Y 625.482,Z 810.371,A -85,B 0,C 180,E1 8401.001,E2 8401.001} C_VEL
LIN {X 0,Y 611.807,Z 782.167,A -85,B 0,C 180,E1 8402.874,E2 8402.874} C_VEL
LIN {X 0,Y 593.208,Z 751.056,A -85,B 0,C 180,E1 8405.162,E2 8405.162} C_VEL
LIN {X 0,Y 593.069,Z 749.56,A -85,B 0,C 180,E1 8405.248,E2 8405.248} C_VEL
LIN {X 0,Y 593.025,Z 749.56,A -85,B 0,C 180,E1 8411.494,E2 8411.494} C_VEL
LIN {X 0,Y 592.993,Z 749.56,A -85,B 0,C 180,E1 8416.518,E2 8416.518} C_VEL
LIN {X 0,Y 592.988,Z 749.56,A -85,B 0,C 180,E1 8422.289,E2 8422.289} C_VEL
LIN {X 0,Y 592.959,Z 749.56,A -85,B 0,C 180,E1 8427.639,E2 8427.639} C_VEL
LIN {X 0,Y 593.054,Z 749.56,A -85,B 0,C 180,E1 8433.104,E2 8433.104} C_VEL
LIN {X 0,Y 593.157,Z 749.56,A -85,B 0,C 180,E1 8439.1,E2 8439.1} C_VEL
LIN {X 0,Y 593.344,Z 749.56,A -85,B 0,C 180,E1 8445.42,E2 8445.42} C_VEL
LIN {X 0,Y 593.689,Z 749.56,A -85,B 0,C 180,E1 8451.211,E2 8451.211} C_VEL
LIN {X 0,Y 593.931,Z 749.56,A -85,B 0,C 180,E1 8457.079,E2 8457.079} C_VEL
LIN {X 0,Y 593.999,Z 749.56,A -85,B 0,C 180,E1 8461.454,E2 8461.454} C_VEL
LIN {X 0,Y 593.706,Z 749.56,A -85,B 0,C 180,E1 8467.308,E2 8467.308} C_VEL
LIN {X 0,Y 593.529,Z 749.56,A -85,B 0,C 180,E1 8473.243,E2 8473.243} C_VEL
LIN {X 0,Y 593.462,Z 749.56,A -85,B 0,C 180,E1 8477.788,E2 8477.788} C_VEL
LIN {X 0,Y 593.316,Z 749.56,A -85,B 0,C 180,E1 8483.523,E2 8483.523} C_VEL
LIN {X 0,Y 593.197,Z 749.56,A -85,B 0,C 180,E1 8488.944,E2 8488.944} C_VEL
LIN {X 0,Y 593.09,Z 749.56,A -85,B 0,C 180,E1 8494.089,E2 8494.089} C_VEL
LIN {X 0,Y 592.989,Z 749.56,A -85,B 0,C 180,E1 8500.137,E2 8500.137} C_VEL
LIN {X 0,Y 593.011,Z 749.56,A -85,B 0,C 180,E1 8500.606,E2 8500.606} C_VEL
LIN {X 0,Y 595.377,Z 755.166,A -85,B 0,C 180,E1 8500.936,E2 8500.936} C_VEL
LIN {X 0,Y 632.035,Z 815.968,A -85,B 0,C 180,E1 8505.214,E2 8505.214} C_VEL
LIN {X 0,Y 633.196,Z 818.024,A -85,B 0,C 180,E1 8505.345,E2 8505.345} C_VEL
LIN {X 0,Y 631.146,Z 864.986,A -85,B 0,C 180,E1 8506.224,E2 8506.224} C_VEL
LIN {X 0,Y 622.735,Z 896.51,A -85,B 0,C 180,E1 8506.607,E2 8506.607} C_VEL
LIN {X 0,Y 622.46,Z 898.539,A -85,B 0,C 180,E1 8506.668,E2 8506.668} C_VEL
LIN {X 0,Y 618.329,Z 940.636,A -85,B 0,C 180,E1 8508.293,E2 8508.293} C_VEL
LIN {X 0,Y 612.824,Z 984.802,A -85,B 0,C 180,E1 8510.575,E2 8510.575} C_VEL
LIN {X 0,Y 606.829,Z 1026.784,A -85,B 0,C 180,E1 8513.404,E2 8513.404} C_VEL
LIN {X 0,Y 600.946,Z 1067.502,A -85,B 0,C 180,E1 8516.913,E2 8516.913} C_VEL
LIN {X 0,Y 595.795,Z 1103.029,A -85,B 0,C 180,E1 8520.791,E2 8520.791} C_VEL
LIN {X 0,Y 591.799,Z 1133.681,A -85,B 0,C 180,E1 8524.968,E2 8524.968} C_VEL
LIN {X 0,Y 588.987,Z 1159.104,A -85,B 0,C 180,E1 8529.377,E2 8529.377} C_VEL
LIN {X 0,Y 587.245,Z 1179.079,A -85,B 0,C 180,E1 8533.827,E2 8533.827} C_VEL
LIN {X 0,Y 586.435,Z 1193.884,A -85,B 0,C 180,E1 8538.276,E2 8538.276} C_VEL
LIN {X 0,Y 586.107,Z 1203.557,A -85,B 0,C 180,E1 8542.593,E2 8542.593} C_VEL
LIN {X 0,Y 586.052,Z 1208.918,A -85,B 0,C 180,E1 8547.043,E2 8547.043} C_VEL
LIN {X 0,Y 586.222,Z 1209.667,A -85,B 0,C 180,E1 8551.476,E2 8551.476} C_VEL
LIN {X 0,Y 586.077,Z 1205.911,A -85,B 0,C 180,E1 8555.919,E2 8555.919} C_VEL
LIN {X 0,Y 586.313,Z 1197.326,A -85,B 0,C 180,E1 8560.393,E2 8560.393} C_VEL
LIN {X 0,Y 587.033,Z 1183.711,A -85,B 0,C 180,E1 8564.916,E2 8564.916} C_VEL
LIN {X 0,Y 588.453,Z 1164.731,A -85,B 0,C 180,E1 8569.501,E2 8569.501} C_VEL
LIN {X 0,Y 590.97,Z 1140.318,A -85,B 0,C 180,E1 8573.969,E2 8573.969} C_VEL
LIN {X 0,Y 594.701,Z 1110.822,A -85,B 0,C 180,E1 8578.245,E2 8578.245} C_VEL
LIN {X 0,Y 599.575,Z 1076.084,A -85,B 0,C 180,E1 8582.226,E2 8582.226} C_VEL
LIN {X 0,Y 605.294,Z 1037.719,A -85,B 0,C 180,E1 8585.743,E2 8585.743} C_VEL
LIN {X 0,Y 611.312,Z 995.639,A -85,B 0,C 180,E1 8588.757,E2 8588.757} C_VEL
LIN {X 0,Y 616.975,Z 951.903,A -85,B 0,C 180,E1 8591.2,E2 8591.2} C_VEL
LIN {X 0,Y 621.738,Z 905.454,A -85,B 0,C 180,E1 8593.107,E2 8593.107} C_VEL
LIN {X 0,Y 625.683,Z 854.86,A -85,B 0,C 180,E1 8594.491,E2 8594.491} C_VEL
LIN {X 0,Y 626.847,Z 820.701,A -85,B 0,C 180,E1 8595.116,E2 8595.116} C_VEL
LIN {X 0,Y 591.395,Z 761.258,A -85,B 0,C 180,E1 8599.353,E2 8599.353} C_VEL
LIN {X 0,Y 585.294,Z 751.37,A -85,B 0,C 180,E1 8600.204,E2 8600.204} C_VEL
LIN {X 0,Y 585.074,Z 749.56,A -85,B 0,C 180,E1 8600.319,E2 8600.319} C_VEL
LIN {X 0,Y 585.104,Z 749.56,A -85,B 0,C 180,E1 8605.735,E2 8605.735} C_VEL
LIN {X 0,Y 585.123,Z 749.56,A -85,B 0,C 180,E1 8611.41,E2 8611.41} C_VEL
LIN {X 0,Y 585.228,Z 749.56,A -85,B 0,C 180,E1 8617.216,E2 8617.216} C_VEL
LIN {X 0,Y 585.448,Z 749.56,A -85,B 0,C 180,E1 8622.748,E2 8622.748} C_VEL
LIN {X 0,Y 585.629,Z 749.56,A -85,B 0,C 180,E1 8628.672,E2 8628.672} C_VEL
LIN {X 0,Y 585.87,Z 749.56,A -85,B 0,C 180,E1 8634.082,E2 8634.082} C_VEL
LIN {X 0,Y 586.067,Z 749.56,A -85,B 0,C 180,E1 8640.004,E2 8640.004} C_VEL
LIN {X 0,Y 585.891,Z 749.56,A -85,B 0,C 180,E1 8644.442,E2 8644.442} C_VEL
LIN {X 0,Y 585.771,Z 749.56,A -85,B 0,C 180,E1 8648.909,E2 8648.909} C_VEL
LIN {X 0,Y 585.474,Z 749.56,A -85,B 0,C 180,E1 8653.437,E2 8653.437} C_VEL
LIN {X 0,Y 585.243,Z 749.56,A -85,B 0,C 180,E1 8659.618,E2 8659.618} C_VEL
LIN {X 0,Y 585.099,Z 749.56,A -85,B 0,C 180,E1 8665.321,E2 8665.321} C_VEL
LIN {X 0,Y 585.063,Z 749.56,A -85,B 0,C 180,E1 8671.108,E2 8671.108} C_VEL
LIN {X 0,Y 585.144,Z 749.675,A -85,B 0,C 180,E1 8675.519,E2 8675.519} C_VEL
LIN {X 0,Y 587.438,Z 755.111,A -85,B 0,C 180,E1 8675.887,E2 8675.887} C_VEL
LIN {X 0,Y 608.247,Z 788.944,A -85,B 0,C 180,E1 8678.744,E2 8678.744} C_VEL
LIN {X 0,Y 620.297,Z 814.712,A -85,B 0,C 180,E1 8680.547,E2 8680.547} C_VEL
LIN {X 0,Y 616.781,Z 858.639,A -85,B 0,C 180,E1 8681.869,E2 8681.869} C_VEL
LIN {X 0,Y 612.405,Z 899.142,A -85,B 0,C 180,E1 8683.62,E2 8683.62} C_VEL
LIN {X 0,Y 606.835,Z 941.387,A -85,B 0,C 180,E1 8686.074,E2 8686.074} C_VEL
LIN {X 0,Y 601.516,Z 978.498,A -85,B 0,C 180,E1 8688.916,E2 8688.916} C_VEL
LIN {X 0,Y 596.127,Z 1017.448,A -85,B 0,C 180,E1 8692.672,E2 8692.672} C_VEL
LIN {X 0,Y 591.99,Z 1050.426,A -85,B 0,C 180,E1 8696.716,E2 8696.716} C_VEL
LIN {X 0,Y 589.091,Z 1077.624,A -85,B 0,C 180,E1 8701.042,E2 8701.042} C_VEL
LIN {X 0,Y 587.332,Z 1098.134,A -85,B 0,C 180,E1 8705.299,E2 8705.299} C_VEL
LIN {X 0,Y 586.541,Z 1112.722,A -85,B 0,C 180,E1 8709.39,E2 8709.39} C_VEL
LIN {X 0,Y 586.027,Z 1122.917,A -85,B 0,C 180,E1 8713.523,E2 8713.523} C_VEL
LIN {X 0,Y 585.794,Z 1128.863,A -85,B 0,C 180,E1 8718.091,E2 8718.091} C_VEL
LIN {X 0,Y 585.96,Z 1129.629,A -85,B 0,C 180,E1 8722.592,E2 8722.592} C_VEL
LIN {X 0,Y 586.158,Z 1125.18,A -85,B 0,C 180,E1 8727.045,E2 8727.045} C_VEL
LIN {X 0,Y 586.377,Z 1115.747,A -85,B 0,C 180,E1 8731.477,E2 8731.477} C_VEL
LIN {X 0,Y 587.104,Z 1102.453,A -85,B 0,C 180,E1 8735.54,E2 8735.54} C_VEL
LIN {X 0,Y 588.562,Z 1082.387,A -85,B 0,C 180,E1 8739.981,E2 8739.981} C_VEL
LIN {X 0,Y 590.995,Z 1058.251,A -85,B 0,C 180,E1 8744.058,E2 8744.058} C_VEL
LIN {X 0,Y 594.926,Z 1027.365,A -85,B 0,C 180,E1 8748.129,E2 8748.129} C_VEL
LIN {X 0,Y 599.572,Z 991.541,A -85,B 0,C 180,E1 8751.824,E2 8751.824} C_VEL
LIN {X 0,Y 604.87,Z 955.278,A -85,B 0,C 180,E1 8754.837,E2 8754.837} C_VEL
LIN {X 0,Y 610.164,Z 916.049,A -85,B 0,C 180,E1 8757.37,E2 8757.37} C_VEL
LIN {X 0,Y 614.904,Z 874.744,A -85,B 0,C 180,E1 8759.39,E2 8759.39} C_VEL
LIN {X 0,Y 619.186,Z 826.762,A -85,B 0,C 180,E1 8761.043,E2 8761.043} C_VEL
LIN {X 0,Y 619.673,Z 813.927,A -85,B 0,C 180,E1 8761.395,E2 8761.395} C_VEL
LIN {X 0,Y 606.814,Z 787.046,A -85,B 0,C 180,E1 8763.238,E2 8763.238} C_VEL
LIN {X 0,Y 585.296,Z 750.997,A -85,B 0,C 180,E1 8765.947,E2 8765.947} C_VEL
LIN {X 0,Y 585.119,Z 749.56,A -85,B 0,C 180,E1 8766.083,E2 8766.083} C_VEL
LIN {X 0,Y 585.119,Z 749.56,A -85,B 0,C 180,E1 8772.182,E2 8772.182} C_VEL
LIN {X 0,Y 585.062,Z 749.56,A -85,B 0,C 180,E1 8777.807,E2 8777.807} C_VEL
LIN {X 0,Y 585.044,Z 749.56,A -85,B 0,C 180,E1 8783.547,E2 8783.547} C_VEL
LIN {X 0,Y 585.038,Z 749.56,A -85,B 0,C 180,E1 8788.891,E2 8788.891} C_VEL
LIN {X 0,Y 585.105,Z 749.56,A -85,B 0,C 180,E1 8794.681,E2 8794.681} C_VEL
LIN {X 0,Y 585.232,Z 749.56,A -85,B 0,C 180,E1 8800.382,E2 8800.382} C_VEL
LIN {X 0,Y 585.469,Z 749.56,A -85,B 0,C 180,E1 8806.563,E2 8806.563} C_VEL
LIN {X 0,Y 585.766,Z 749.56,A -85,B 0,C 180,E1 8811.091,E2 8811.091} C_VEL
LIN {X 0,Y 586.021,Z 749.56,A -85,B 0,C 180,E1 8817.04,E2 8817.04} C_VEL
LIN {X 0,Y 586.091,Z 749.56,A -85,B 0,C 180,E1 8821.473,E2 8821.473} C_VEL
LIN {X 0,Y 585.792,Z 749.56,A -85,B 0,C 180,E1 8827.407,E2 8827.407} C_VEL
LIN {X 0,Y 585.625,Z 749.56,A -85,B 0,C 180,E1 8833.425,E2 8833.425} C_VEL
LIN {X 0,Y 585.548,Z 749.56,A -85,B 0,C 180,E1 8838.036,E2 8838.036} C_VEL
LIN {X 0,Y 585.387,Z 749.56,A -85,B 0,C 180,E1 8842.777,E2 8842.777} C_VEL
LIN {X 0,Y 585.302,Z 749.56,A -85,B 0,C 180,E1 8848.619,E2 8848.619} C_VEL
LIN {X 0,Y 585.165,Z 749.56,A -85,B 0,C 180,E1 8854.616,E2 8854.616} C_VEL
LIN {X 0,Y 585.091,Z 749.643,A -85,B 0,C 180,E1 8859.812,E2 8859.812} C_VEL
LIN {X 0,Y 587.524,Z 755.23,A -85,B 0,C 180,E1 8860.156,E2 8860.156} C_VEL
LIN {X 0,Y 623.294,Z 814.311,A -85,B 0,C 180,E1 8864.461,E2 8864.461} C_VEL
LIN {X 0,Y 627.121,Z 821.115,A -85,B 0,C 180,E1 8864.902,E2 8864.902} C_VEL
LIN {X 0,Y 624.533,Z 873.813,A -85,B 0,C 180,E1 8865.958,E2 8865.958} C_VEL
LIN {X 0,Y 622.46,Z 898.539,A -85,B 0,C 180,E1 8866.668,E2 8866.668} C_VEL
LIN {X 0,Y 617.795,Z 915.545,A -85,B 0,C 180,E1 8867.007,E2 8867.007} C_VEL
LIN {X 0,Y 613.212,Z 931.376,A -85,B 0,C 180,E1 8867.398,E2 8867.398} C_VEL
LIN {X 0,Y 608.037,Z 973.454,A -85,B 0,C 180,E1 8869.426,E2 8869.426} C_VEL
LIN {X 0,Y 601.361,Z 1019.332,A -85,B 0,C 180,E1 8872.369,E2 8872.369} C_VEL
LIN {X 0,Y 595.313,Z 1059.002,A -85,B 0,C 180,E1 8875.671,E2 8875.671} C_VEL
LIN {X 0,Y 589.65,Z 1096.43,A -85,B 0,C 180,E1 8879.592,E2 8879.592} C_VEL
LIN {X 0,Y 584.95,Z 1129.131,A -85,B 0,C 180,E1 8883.948,E2 8883.948} C_VEL
LIN {X 0,Y 581.785,Z 1154.987,A -85,B 0,C 180,E1 8888.276,E2 8888.276} C_VEL
LIN {X 0,Y 579.722,Z 1176.512,A -85,B 0,C 180,E1 8892.958,E2 8892.958} C_VEL
